LIN {X 0,Y 256.282,Z 675.842,A -85,B 0,C 180,E1 -18466.303,E2 -18466.303} C_VEL
LIN {X 0,Y 258.512,Z 670.213,A -85,B 0,C 180,E1 -18469.867,E2 -18469.867} C_VEL
LIN {X 0,Y 261.173,Z 664.065,A -85,B 0,C 180,E1 -18472.966,E2 -18472.966} C_VEL
LIN {X 0,Y 264.928,Z 655.56,A -85,B 0,C 180,E1 -18476.382,E2 -18476.382} C_VEL
LIN {X 0,Y 269.071,Z 646.458,A -85,B 0,C 180,E1 -18479.324,E2 -18479.324} C_VEL
LIN {X 0,Y 273.55,Z 636.336,A -85,B 0,C 180,E1 -18482.025,E2 -18482.025} C_VEL
LIN {X 0,Y 278.615,Z 624.618,A -85,B 0,C 180,E1 -18484.58,E2 -18484.58} C_VEL
LIN {X 0,Y 283.109,Z 613.564,A -85,B 0,C 180,E1 -18486.569,E2 -18486.569} C_VEL
LIN {X 0,Y 287.912,Z 600.645,A -85,B 0,C 180,E1 -18488.505,E2 -18488.505} C_VEL
LIN {X 0,Y 292.653,Z 586.785,A -85,B 0,C 180,E1 -18490.196,E2 -18490.196} C_VEL
LIN {X 0,Y 296.833,Z 573.328,A -85,B 0,C 180,E1 -18491.525,E2 -18491.525} C_VEL
LIN {X 0,Y 300.553,Z 558.842,A -85,B 0,C 180,E1 -18492.697,E2 -18492.697} C_VEL
LIN {X 0,Y 303.97,Z 543.205,A -85,B 0,C 180,E1 -18493.688,E2 -18493.688} C_VEL
LIN {X 0,Y 306.838,Z 526.737,A -85,B 0,C 180,E1 -18494.466,E2 -18494.466} C_VEL
LIN {X 0,Y 308.914,Z 510.285,A -85,B 0,C 180,E1 -18495.012,E2 -18495.012} C_VEL
LIN {X 0,Y 316.401,Z 389.403,A -85,B 0,C 180,E1 -18497.751,E2 -18497.751} C_VEL
LIN {X 0,Y 310.716,Z 378.003,A -85,B 0,C 180,E1 -18499.592,E2 -18499.592} C_VEL
LIN {X 0,Y 304.506,Z 366.741,A -85,B 0,C 180,E1 -18501.741,E2 -18501.741} C_VEL
LIN {X 0,Y 298.717,Z 357.161,A -85,B 0,C 180,E1 -18503.921,E2 -18503.921} C_VEL
LIN {X 0,Y 292.889,Z 347.944,A -85,B 0,C 180,E1 -18506.349,E2 -18506.349} C_VEL
LIN {X 0,Y 289.275,Z 342.774,A -85,B 0,C 180,E1 -18507.981,E2 -18507.981} C_VEL
LIN {X 0,Y 285.853,Z 337.855,A -85,B 0,C 180,E1 -18509.676,E2 -18509.676} C_VEL
LIN {X 0,Y 281.014,Z 331.224,A -85,B 0,C 180,E1 -18512.335,E2 -18512.335} C_VEL
LIN {X 0,Y 278.285,Z 328.209,A -85,B 0,C 180,E1 -18513.973,E2 -18513.973} C_VEL
LIN {X 0,Y 277.263,Z 326.406,A -85,B 0,C 180,E1 -18514.686,E2 -18514.686} C_VEL
LIN {X 0,Y 274.465,Z 324.032,A -85,B 0,C 180,E1 -18516.597,E2 -18516.597} C_VEL
LIN {X 0,Y 272.679,Z 320.875,A -85,B 0,C 180,E1 -18518.104,E2 -18518.104} C_VEL
LIN {X 0,Y 269.81,Z 318.889,A -85,B 0,C 180,E1 -18520.579,E2 -18520.579} C_VEL
LIN {X 0,Y 268.115,Z 316.082,A -85,B 0,C 180,E1 -18522.567,E2 -18522.567} C_VEL
LIN {X 0,Y 267.662,Z 314.997,A -85,B 0,C 180,E1 -18523.213,E2 -18523.213} C_VEL
LIN {X 0,Y 263.908,Z 312.436,A -85,B 0,C 180,E1 -18530.033,E2 -18530.033} C_VEL
LIN {X 0,Y 263.493,Z 311.642,A -85,B 0,C 180,E1 -18532.337,E2 -18532.337} C_VEL
LIN {X 0,Y 263.433,Z 311.699,A -85,B 0,C 180,E1 -18534.643,E2 -18534.643} C_VEL
LIN {X 0,Y 264.572,Z 312.819,A -85,B 0,C 180,E1 -18539.24,E2 -18539.24} C_VEL
LIN {X 0,Y 268.053,Z 315.309,A -85,B 0,C 180,E1 -18544.706,E2 -18544.706} C_VEL
LIN {X 0,Y 269.415,Z 318.063,A -85,B 0,C 180,E1 -18546.413,E2 -18546.413} C_VEL
LIN {X 0,Y 272.147,Z 320.485,A -85,B 0,C 180,E1 -18548.914,E2 -18548.914} C_VEL
LIN {X 0,Y 272.948,Z 321.205,A -85,B 0,C 180,E1 -18549.565,E2 -18549.565} C_VEL
LIN {X 0,Y 274.825,Z 324.302,A -85,B 0,C 180,E1 -18551.105,E2 -18551.105} C_VEL
LIN {X 0,Y 277.54,Z 326.712,A -85,B 0,C 180,E1 -18552.942,E2 -18552.942} C_VEL
LIN {X 0,Y 279.846,Z 330.125,A -85,B 0,C 180,E1 -18554.441,E2 -18554.441} C_VEL
LIN {X 0,Y 281.946,Z 332.247,A -85,B 0,C 180,E1 -18555.636,E2 -18555.636} C_VEL
LIN {X 0,Y 284.858,Z 335.997,A -85,B 0,C 180,E1 -18557.222,E2 -18557.222} C_VEL
LIN {X 0,Y 286.192,Z 337.735,A -85,B 0,C 180,E1 -18557.908,E2 -18557.908} C_VEL
LIN {X 0,Y 290.002,Z 342.639,A -85,B 0,C 180,E1 -18559.742,E2 -18559.742} C_VEL
LIN {X 0,Y 294.08,Z 348.095,A -85,B 0,C 180,E1 -18561.53,E2 -18561.53} C_VEL
LIN {X 0,Y 299.43,Z 355.459,A -85,B 0,C 180,E1 -18563.674,E2 -18563.674} C_VEL
LIN {X 0,Y 306.714,Z 366.264,A -85,B 0,C 180,E1 -18566.307,E2 -18566.307} C_VEL
LIN {X 0,Y 313.655,Z 377.566,A -85,B 0,C 180,E1 -18568.583,E2 -18568.583} C_VEL
LIN {X 0,Y 316.643,Z 382.91,A -85,B 0,C 180,E1 -18569.512,E2 -18569.512} C_VEL
LIN {X 0,Y 315.495,Z 402.823,A -85,B 0,C 180,E1 -18569.977,E2 -18569.977} C_VEL
LIN {X 0,Y 309.458,Z 498.844,A -85,B 0,C 180,E1 -18572.149,E2 -18572.149} C_VEL
LIN {X 0,Y 307.487,Z 515.059,A -85,B 0,C 180,E1 -18572.712,E2 -18572.712} C_VEL
LIN {X 0,Y 304.889,Z 531.096,A -85,B 0,C 180,E1 -18573.517,E2 -18573.517} C_VEL
LIN {X 0,Y 301.499,Z 547.393,A -85,B 0,C 180,E1 -18574.599,E2 -18574.599} C_VEL
LIN {X 0,Y 297.861,Z 561.75,A -85,B 0,C 180,E1 -18575.799,E2 -18575.799} C_VEL
LIN {X 0,Y 293.557,Z 576.25,A -85,B 0,C 180,E1 -18577.304,E2 -18577.304} C_VEL
LIN {X 0,Y 289.209,Z 589.149,A -85,B 0,C 180,E1 -18578.956,E2 -18578.956} C_VEL
LIN {X 0,Y 284.196,Z 602.561,A -85,B 0,C 180,E1 -18581.04,E2 -18581.04} C_VEL
LIN {X 0,Y 279.535,Z 613.986,A -85,B 0,C 180,E1 -18583.188,E2 -18583.188} C_VEL
LIN {X 0,Y 274.591,Z 625.334,A -85,B 0,C 180,E1 -18585.779,E2 -18585.779} C_VEL
LIN {X 0,Y 270.165,Z 634.852,A -85,B 0,C 180,E1 -18588.444,E2 -18588.444} C_VEL
LIN {X 0,Y 266.327,Z 642.967,A -85,B 0,C 180,E1 -18591.19,E2 -18591.19} C_VEL
LIN {X 0,Y 263.087,Z 649.861,A -85,B 0,C 180,E1 -18594.006,E2 -18594.006} C_VEL
LIN {X 0,Y 260.017,Z 656.29,A -85,B 0,C 180,E1 -18597.277,E2 -18597.277} C_VEL
LIN {X 0,Y 257.501,Z 661.786,A -85,B 0,C 180,E1 -18600.856,E2 -18600.856} C_VEL
LIN {X 0,Y 255.936,Z 665.412,A -85,B 0,C 180,E1 -18603.937,E2 -18603.937} C_VEL
LIN {X 0,Y 254.774,Z 668.176,A -85,B 0,C 180,E1 -18607.282,E2 -18607.282} C_VEL
LIN {X 0,Y 254.125,Z 669.944,A -85,B 0,C 180,E1 -18610.618,E2 -18610.618} C_VEL
LIN {X 0,Y 253.789,Z 670.613,A -85,B 0,C 180,E1 -18613.923,E2 -18613.923} C_VEL
LIN {X 0,Y 253.738,Z 670.334,A -85,B 0,C 180,E1 -18617.198,E2 -18617.198} C_VEL
LIN {X 0,Y 253.774,Z 669.044,A -85,B 0,C 180,E1 -18620.435,E2 -18620.435} C_VEL
LIN {X 0,Y 254.305,Z 666.26,A -85,B 0,C 180,E1 -18624.221,E2 -18624.221} C_VEL
LIN {X 0,Y 254.766,Z 662.566,A -85,B 0,C 180,E1 -18627.628,E2 -18627.628} C_VEL
LIN {X 0,Y 255.672,Z 657.991,A -85,B 0,C 180,E1 -18630.787,E2 -18630.787} C_VEL
LIN {X 0,Y 257.085,Z 652.288,A -85,B 0,C 180,E1 -18633.919,E2 -18633.919} C_VEL
LIN {X 0,Y 258.941,Z 645.419,A -85,B 0,C 180,E1 -18637.015,E2 -18637.015} C_VEL
LIN {X 0,Y 261.842,Z 635.962,A -85,B 0,C 180,E1 -18640.438,E2 -18640.438} C_VEL
LIN {X 0,Y 265.051,Z 625.811,A -85,B 0,C 180,E1 -18643.415,E2 -18643.415} C_VEL
LIN {X 0,Y 268.266,Z 615.356,A -85,B 0,C 180,E1 -18645.966,E2 -18645.966} C_VEL
LIN {X 0,Y 271.802,Z 603.133,A -85,B 0,C 180,E1 -18648.466,E2 -18648.466} C_VEL
LIN {X 0,Y 275.208,Z 590.86,A -85,B 0,C 180,E1 -18650.557,E2 -18650.557} C_VEL
LIN {X 0,Y 278.588,Z 577.562,A -85,B 0,C 180,E1 -18652.43,E2 -18652.43} C_VEL
LIN {X 0,Y 281.942,Z 563.146,A -85,B 0,C 180,E1 -18654.09,E2 -18654.09} C_VEL
LIN {X 0,Y 284.627,Z 549.4,A -85,B 0,C 180,E1 -18655.405,E2 -18655.405} C_VEL
LIN {X 0,Y 286.727,Z 536.983,A -85,B 0,C 180,E1 -18656.376,E2 -18656.376} C_VEL
LIN {X 0,Y 289.155,Z 520.691,A -85,B 0,C 180,E1 -18657.356,E2 -18657.356} C_VEL
LIN {X 0,Y 290.872,Z 504.966,A -85,B 0,C 180,E1 -18658.06,E2 -18658.06} C_VEL
LIN {X 0,Y 292.168,Z 487.884,A -85,B 0,C 180,E1 -18658.56,E2 -18658.56} C_VEL
LIN {X 0,Y 297.829,Z 371.285,A -85,B 0,C 180,E1 -18661.275,E2 -18661.275} C_VEL
LIN {X 0,Y 297.355,Z 369.401,A -85,B 0,C 180,E1 -18661.409,E2 -18661.409} C_VEL
LIN {X 0,Y 291.594,Z 358.102,A -85,B 0,C 180,E1 -18662.726,E2 -18662.726} C_VEL
LIN {X 0,Y 282.106,Z 341.691,A -85,B 0,C 180,E1 -18664.988,E2 -18664.988} C_VEL
LIN {X 0,Y 273.66,Z 328.4,A -85,B 0,C 180,E1 -18667.161,E2 -18667.161} C_VEL
LIN {X 0,Y 265.648,Z 316.865,A -85,B 0,C 180,E1 -18669.382,E2 -18669.382} C_VEL
LIN {X 0,Y 262.439,Z 312.49,A -85,B 0,C 180,E1 -18670.328,E2 -18670.328} C_VEL
LIN {X 0,Y 260.022,Z 309.315,A -85,B 0,C 180,E1 -18671.062,E2 -18671.062} C_VEL
LIN {X 0,Y 259.132,Z 307.907,A -85,B 0,C 180,E1 -18671.349,E2 -18671.349} C_VEL
LIN {X 0,Y 256.924,Z 305.562,A -85,B 0,C 180,E1 -18672.024,E2 -18672.024} C_VEL
LIN {X 0,Y 256.02,Z 302.892,A -85,B 0,C 180,E1 -18672.413,E2 -18672.413} C_VEL
LIN {X 0,Y 256.005,Z 302.89,A -85,B 0,C 180,E1 -18676.66,E2 -18676.66} C_VEL
LIN {X 0,Y 256.044,Z 302.866,A -85,B 0,C 180,E1 -18680.852,E2 -18680.852} C_VEL
LIN {X 0,Y 256.042,Z 302.843,A -85,B 0,C 180,E1 -18682.1,E2 -18682.1} C_VEL
LIN {X 0,Y 255.418,Z 302.915,A -85,B 0,C 180,E1 -18683.412,E2 -18683.412} C_VEL
LIN {X 0,Y 252.558,Z 303.294,A -85,B 0,C 180,E1 -18685.55,E2 -18685.55} C_VEL
LIN {X 0,Y 250.108,Z 303.636,A -85,B 0,C 180,E1 -18687.29,E2 -18687.29} C_VEL
LIN {X 0,Y 249.065,Z 303.772,A -85,B 0,C 180,E1 -18688.641,E2 -18688.641} C_VEL
LIN {X 0,Y 248.987,Z 303.771,A -85,B 0,C 180,E1 -18689.099,E2 -18689.099} C_VEL
LIN {X 0,Y 249.031,Z 303.776,A -85,B 0,C 180,E1 -18693.156,E2 -18693.156} C_VEL
LIN {X 0,Y 249.055,Z 303.753,A -85,B 0,C 180,E1 -18696.729,E2 -18696.729} C_VEL
LIN {X 0,Y 249.087,Z 303.765,A -85,B 0,C 180,E1 -18700.209,E2 -18700.209} C_VEL
LIN {X 0,Y 249.197,Z 303.744,A -85,B 0,C 180,E1 -18703.618,E2 -18703.618} C_VEL
LIN {X 0,Y 249.244,Z 303.728,A -85,B 0,C 180,E1 -18708.615,E2 -18708.615} C_VEL
LIN {X 0,Y 249.445,Z 303.723,A -85,B 0,C 180,E1 -18711.901,E2 -18711.901} C_VEL
LIN {X 0,Y 249.279,Z 303.725,A -85,B 0,C 180,E1 -18715.147,E2 -18715.147} C_VEL
LIN {X 0,Y 249.672,Z 303.691,A -85,B 0,C 180,E1 -18718.386,E2 -18718.386} C_VEL
LIN {X 0,Y 249.675,Z 303.679,A -85,B 0,C 180,E1 -18721.612,E2 -18721.612} C_VEL
LIN {X 0,Y 249.449,Z 303.691,A -85,B 0,C 180,E1 -18726.47,E2 -18726.47} C_VEL
LIN {X 0,Y 249.343,Z 303.732,A -85,B 0,C 180,E1 -18729.736,E2 -18729.736} C_VEL
LIN {X 0,Y 249.183,Z 303.759,A -85,B 0,C 180,E1 -18734.704,E2 -18734.704} C_VEL
LIN {X 0,Y 249.12,Z 303.767,A -85,B 0,C 180,E1 -18738.078,E2 -18738.078} C_VEL
LIN {X 0,Y 249.086,Z 303.769,A -85,B 0,C 180,E1 -18741.517,E2 -18741.517} C_VEL
LIN {X 0,Y 249.129,Z 303.763,A -85,B 0,C 180,E1 -18745.481,E2 -18745.481} C_VEL
LIN {X 0,Y 249.079,Z 303.772,A -85,B 0,C 180,E1 -18748.991,E2 -18748.991} C_VEL
LIN {X 0,Y 249.026,Z 303.779,A -85,B 0,C 180,E1 -18752.285,E2 -18752.285} C_VEL
LIN {X 0,Y 249.973,Z 306.545,A -85,B 0,C 180,E1 -18752.706,E2 -18752.706} C_VEL
LIN {X 0,Y 252.086,Z 308.765,A -85,B 0,C 180,E1 -18753.408,E2 -18753.408} C_VEL
LIN {X 0,Y 252.84,Z 309.519,A -85,B 0,C 180,E1 -18753.654,E2 -18753.654} C_VEL
LIN {X 0,Y 254.89,Z 312.734,A -85,B 0,C 180,E1 -18754.358,E2 -18754.358} C_VEL
LIN {X 0,Y 256.51,Z 314.52,A -85,B 0,C 180,E1 -18754.867,E2 -18754.867} C_VEL
LIN {X 0,Y 259.22,Z 318.185,A -85,B 0,C 180,E1 -18755.722,E2 -18755.722} C_VEL
LIN {X 0,Y 264.025,Z 325.444,A -85,B 0,C 180,E1 -18757.19,E2 -18757.19} C_VEL
LIN {X 0,Y 270.599,Z 336.395,A -85,B 0,C 180,E1 -18759.096,E2 -18759.096} C_VEL
LIN {X 0,Y 278.225,Z 350.18,A -85,B 0,C 180,E1 -18761.173,E2 -18761.173} C_VEL
LIN {X 0,Y 285.454,Z 364.869,A -85,B 0,C 180,E1 -18763.034,E2 -18763.034} C_VEL
LIN {X 0,Y 292.165,Z 379.915,A -85,B 0,C 180,E1 -18764.686,E2 -18764.686} C_VEL
LIN {X 0,Y 285.516,Z 510.664,A -85,B 0,C 180,E1 -18767.806,E2 -18767.806} C_VEL
LIN {X 0,Y 283.759,Z 527.699,A -85,B 0,C 180,E1 -18768.448,E2 -18768.448} C_VEL
LIN {X 0,Y 281.493,Z 543.45,A -85,B 0,C 180,E1 -18769.288,E2 -18769.288} C_VEL
LIN {X 0,Y 278.588,Z 559.632,A -85,B 0,C 180,E1 -18770.433,E2 -18770.433} C_VEL
LIN {X 0,Y 275.831,Z 572.821,A -85,B 0,C 180,E1 -18771.607,E2 -18771.607} C_VEL
LIN {X 0,Y 272.213,Z 587.811,A -85,B 0,C 180,E1 -18773.263,E2 -18773.263} C_VEL
LIN {X 0,Y 268.642,Z 601.267,A -85,B 0,C 180,E1 -18775.091,E2 -18775.091} C_VEL
LIN {X 0,Y 265.222,Z 613.539,A -85,B 0,C 180,E1 -18777.097,E2 -18777.097} C_VEL
LIN {X 0,Y 261.658,Z 624.974,A -85,B 0,C 180,E1 -18779.314,E2 -18779.314} C_VEL
LIN {X 0,Y 258.167,Z 636.389,A -85,B 0,C 180,E1 -18781.992,E2 -18781.992} C_VEL
LIN {X 0,Y 255.048,Z 646.135,A -85,B 0,C 180,E1 -18784.716,E2 -18784.716} C_VEL
LIN {X 0,Y 252.296,Z 655.591,A -85,B 0,C 180,E1 -18787.91,E2 -18787.91} C_VEL
LIN {X 0,Y 250.074,Z 663.425,A -85,B 0,C 180,E1 -18791.144,E2 -18791.144} C_VEL
LIN {X 0,Y 248.522,Z 670.114,A -85,B 0,C 180,E1 -18794.558,E2 -18794.558} C_VEL
LIN {X 0,Y 247.555,Z 675.124,A -85,B 0,C 180,E1 -18797.707,E2 -18797.707} C_VEL
LIN {X 0,Y 247.097,Z 678.259,A -85,B 0,C 180,E1 -18800.174,E2 -18800.174} C_VEL
LIN {X 0,Y 246.938,Z 681.534,A -85,B 0,C 180,E1 -18803.463,E2 -18803.463} C_VEL
LIN {X 0,Y 246.885,Z 683.72,A -85,B 0,C 180,E1 -18806.736,E2 -18806.736} C_VEL
LIN {X 0,Y 246.981,Z 684.942,A -85,B 0,C 180,E1 -18810,E2 -18810} C_VEL
LIN {X 0,Y 246.837,Z 685.129,A -85,B 0,C 180,E1 -18813.265,E2 -18813.265} C_VEL
LIN {X 0,Y 246.86,Z 684.395,A -85,B 0,C 180,E1 -18816.539,E2 -18816.539} C_VEL
LIN {X 0,Y 247.156,Z 682.668,A -85,B 0,C 180,E1 -18819.824,E2 -18819.824} C_VEL
LIN {X 0,Y 247.92,Z 680.007,A -85,B 0,C 180,E1 -18823.108,E2 -18823.108} C_VEL
LIN {X 0,Y 249.271,Z 676.096,A -85,B 0,C 180,E1 -18826.547,E2 -18826.547} C_VEL
LIN {X 0,Y 251.161,Z 671.616,A -85,B 0,C 180,E1 -18829.621,E2 -18829.621} C_VEL
LIN {X 0,Y 253.819,Z 665.734,A -85,B 0,C 180,E1 -18832.808,E2 -18832.808} C_VEL
LIN {X 0,Y 257.555,Z 657.691,A -85,B 0,C 180,E1 -18836.322,E2 -18836.322} C_VEL
LIN {X 0,Y 261.714,Z 649.102,A -85,B 0,C 180,E1 -18839.346,E2 -18839.346} C_VEL
LIN {X 0,Y 266.735,Z 638.415,A -85,B 0,C 180,E1 -18842.392,E2 -18842.392} C_VEL
LIN {X 0,Y 272.066,Z 626.675,A -85,B 0,C 180,E1 -18845.083,E2 -18845.083} C_VEL
LIN {X 0,Y 276.631,Z 615.951,A -85,B 0,C 180,E1 -18847.113,E2 -18847.113} C_VEL
LIN {X 0,Y 281.946,Z 602.57,A -85,B 0,C 180,E1 -18849.209,E2 -18849.209} C_VEL
LIN {X 0,Y 286.428,Z 590.233,A -85,B 0,C 180,E1 -18850.79,E2 -18850.79} C_VEL
LIN {X 0,Y 291.079,Z 575.761,A -85,B 0,C 180,E1 -18852.302,E2 -18852.302} C_VEL
LIN {X 0,Y 295.442,Z 559.974,A -85,B 0,C 180,E1 -18853.619,E2 -18853.619} C_VEL
LIN {X 0,Y 298.693,Z 546.026,A -85,B 0,C 180,E1 -18854.545,E2 -18854.545} C_VEL
LIN {X 0,Y 301.828,Z 529.373,A -85,B 0,C 180,E1 -18855.376,E2 -18855.376} C_VEL
LIN {X 0,Y 304.023,Z 513.672,A -85,B 0,C 180,E1 -18855.918,E2 -18855.918} C_VEL
LIN {X 0,Y 305.657,Z 491.795,A -85,B 0,C 180,E1 -18856.48,E2 -18856.48} C_VEL
LIN {X 0,Y 311.962,Z 392.471,A -85,B 0,C 180,E1 -18858.712,E2 -18858.712} C_VEL
LIN {X 0,Y 306.688,Z 381.757,A -85,B 0,C 180,E1 -18860.508,E2 -18860.508} C_VEL
LIN {X 0,Y 300.287,Z 370.018,A -85,B 0,C 180,E1 -18862.844,E2 -18862.844} C_VEL
LIN {X 0,Y 294.471,Z 360.375,A -85,B 0,C 180,E1 -18865.173,E2 -18865.173} C_VEL
LIN {X 0,Y 289.954,Z 353.204,A -85,B 0,C 180,E1 -18867.158,E2 -18867.158} C_VEL
LIN {X 0,Y 287.239,Z 349.171,A -85,B 0,C 180,E1 -18868.442,E2 -18868.442} C_VEL
LIN {X 0,Y 283.9,Z 344.285,A -85,B 0,C 180,E1 -18870.147,E2 -18870.147} C_VEL
LIN {X 0,Y 279.285,Z 337.821,A -85,B 0,C 180,E1 -18872.764,E2 -18872.764} C_VEL
LIN {X 0,Y 276.497,Z 334.578,A -85,B 0,C 180,E1 -18874.505,E2 -18874.505} C_VEL
LIN {X 0,Y 275.556,Z 333.045,A -85,B 0,C 180,E1 -18875.176,E2 -18875.176} C_VEL
LIN {X 0,Y 272.747,Z 330.381,A -85,B 0,C 180,E1 -18877.191,E2 -18877.191} C_VEL
LIN {X 0,Y 271.223,Z 327.703,A -85,B 0,C 180,E1 -18878.525,E2 -18878.525} C_VEL
LIN {X 0,Y 268.356,Z 325.445,A -85,B 0,C 180,E1 -18881.14,E2 -18881.14} C_VEL
LIN {X 0,Y 266.807,Z 322.608,A -85,B 0,C 180,E1 -18883.09,E2 -18883.09} C_VEL
LIN {X 0,Y 266.581,Z 321.964,A -85,B 0,C 180,E1 -18883.44,E2 -18883.44} C_VEL
LIN {X 0,Y 262.982,Z 319.422,A -85,B 0,C 180,E1 -18890.208,E2 -18890.208} C_VEL
LIN {X 0,Y 262.617,Z 318.699,A -85,B 0,C 180,E1 -18892.311,E2 -18892.311} C_VEL
LIN {X 0,Y 262.557,Z 318.73,A -85,B 0,C 180,E1 -18894.625,E2 -18894.625} C_VEL
LIN {X 0,Y 263.687,Z 319.881,A -85,B 0,C 180,E1 -18899.237,E2 -18899.237} C_VEL
LIN {X 0,Y 266.881,Z 322.267,A -85,B 0,C 180,E1 -18904.389,E2 -18904.389} C_VEL
LIN {X 0,Y 268.387,Z 325.133,A -85,B 0,C 180,E1 -18906.296,E2 -18906.296} C_VEL
LIN {X 0,Y 271.018,Z 327.446,A -85,B 0,C 180,E1 -18908.741,E2 -18908.741} C_VEL
LIN {X 0,Y 271.498,Z 327.944,A -85,B 0,C 180,E1 -18909.147,E2 -18909.147} C_VEL
LIN {X 0,Y 273.536,Z 331.203,A -85,B 0,C 180,E1 -18910.853,E2 -18910.853} C_VEL
LIN {X 0,Y 275.971,Z 333.473,A -85,B 0,C 180,E1 -18912.549,E2 -18912.549} C_VEL
LIN {X 0,Y 278.466,Z 337.018,A -85,B 0,C 180,E1 -18914.199,E2 -18914.199} C_VEL
LIN {X 0,Y 280.138,Z 338.785,A -85,B 0,C 180,E1 -18915.179,E2 -18915.179} C_VEL
LIN {X 0,Y 283.249,Z 342.749,A -85,B 0,C 180,E1 -18916.912,E2 -18916.912} C_VEL
LIN {X 0,Y 287.981,Z 349.137,A -85,B 0,C 180,E1 -18919.3,E2 -18919.3} C_VEL
LIN {X 0,Y 292.559,Z 355.305,A -85,B 0,C 180,E1 -18921.353,E2 -18921.353} C_VEL
LIN {X 0,Y 299.18,Z 364.828,A -85,B 0,C 180,E1 -18924.025,E2 -18924.025} C_VEL
LIN {X 0,Y 306.111,Z 375.653,A -85,B 0,C 180,E1 -18926.53,E2 -18926.53} C_VEL
LIN {X 0,Y 312.261,Z 386.159,A -85,B 0,C 180,E1 -18928.565,E2 -18928.565} C_VEL
LIN {X 0,Y 304.942,Z 498.932,A -85,B 0,C 180,E1 -18931.126,E2 -18931.126} C_VEL
LIN {X 0,Y 302.876,Z 515.219,A -85,B 0,C 180,E1 -18931.685,E2 -18931.685} C_VEL
LIN {X 0,Y 300.358,Z 530.516,A -85,B 0,C 180,E1 -18932.454,E2 -18932.454} C_VEL
LIN {X 0,Y 297.394,Z 544.888,A -85,B 0,C 180,E1 -18933.385,E2 -18933.385} C_VEL
LIN {X 0,Y 294.011,Z 558.094,A -85,B 0,C 180,E1 -18934.443,E2 -18934.443} C_VEL
LIN {X 0,Y 289.61,Z 572.976,A -85,B 0,C 180,E1 -18935.919,E2 -18935.919} C_VEL
LIN {X 0,Y 284.973,Z 586.716,A -85,B 0,C 180,E1 -18937.602,E2 -18937.602} C_VEL
LIN {X 0,Y 280.132,Z 599.542,A -85,B 0,C 180,E1 -18939.514,E2 -18939.514} C_VEL
LIN {X 0,Y 274.408,Z 613.211,A -85,B 0,C 180,E1 -18942.035,E2 -18942.035} C_VEL
LIN {X 0,Y 269.135,Z 624.8,A -85,B 0,C 180,E1 -18944.689,E2 -18944.689} C_VEL
LIN {X 0,Y 264.526,Z 634.308,A -85,B 0,C 180,E1 -18947.352,E2 -18947.352} C_VEL
LIN {X 0,Y 259.896,Z 643.608,A -85,B 0,C 180,E1 -18950.544,E2 -18950.544} C_VEL
LIN {X 0,Y 256.07,Z 651.292,A -85,B 0,C 180,E1 -18953.837,E2 -18953.837} C_VEL
LIN {X 0,Y 252.928,Z 657.539,A -85,B 0,C 180,E1 -18957.191,E2 -18957.191} C_VEL
LIN {X 0,Y 250.04,Z 663.516,A -85,B 0,C 180,E1 -18961.456,E2 -18961.456} C_VEL
LIN {X 0,Y 248.499,Z 666.914,A -85,B 0,C 180,E1 -18964.898,E2 -18964.898} C_VEL
LIN {X 0,Y 247.442,Z 669.272,A -85,B 0,C 180,E1 -18968.331,E2 -18968.331} C_VEL
LIN {X 0,Y 246.86,Z 670.552,A -85,B 0,C 180,E1 -18971.75,E2 -18971.75} C_VEL
LIN {X 0,Y 246.689,Z 670.77,A -85,B 0,C 180,E1 -18975.616,E2 -18975.616} C_VEL
LIN {X 0,Y 246.63,Z 670.118,A -85,B 0,C 180,E1 -18978.494,E2 -18978.494} C_VEL
LIN {X 0,Y 246.799,Z 668.406,A -85,B 0,C 180,E1 -18981.814,E2 -18981.814} C_VEL
LIN {X 0,Y 247.291,Z 665.747,A -85,B 0,C 180,E1 -18985.109,E2 -18985.109} C_VEL
LIN {X 0,Y 248.112,Z 660.959,A -85,B 0,C 180,E1 -18989.188,E2 -18989.188} C_VEL
LIN {X 0,Y 249.236,Z 655.904,A -85,B 0,C 180,E1 -18992.424,E2 -18992.424} C_VEL
LIN {X 0,Y 250.922,Z 649.748,A -85,B 0,C 180,E1 -18995.626,E2 -18995.626} C_VEL
LIN {X 0,Y 253.494,Z 641.227,A -85,B 0,C 180,E1 -18999.173,E2 -18999.173} C_VEL
LIN {X 0,Y 256.533,Z 632.019,A -85,B 0,C 180,E1 -19002.258,E2 -19002.258} C_VEL
LIN {X 0,Y 259.573,Z 622.575,A -85,B 0,C 180,E1 -19004.905,E2 -19004.905} C_VEL
LIN {X 0,Y 263.032,Z 611.599,A -85,B 0,C 180,E1 -19007.493,E2 -19007.493} C_VEL
LIN {X 0,Y 266.843,Z 598.664,A -85,B 0,C 180,E1 -19010.022,E2 -19010.022} C_VEL
LIN {X 0,Y 270.777,Z 584.323,A -85,B 0,C 180,E1 -19012.308,E2 -19012.308} C_VEL
LIN {X 0,Y 274.498,Z 569.698,A -85,B 0,C 180,E1 -19014.183,E2 -19014.183} C_VEL
LIN {X 0,Y 277.646,Z 555.32,A -85,B 0,C 180,E1 -19015.689,E2 -19015.689} C_VEL
LIN {X 0,Y 280.462,Z 539.768,A -85,B 0,C 180,E1 -19017.013,E2 -19017.013} C_VEL
LIN {X 0,Y 283.069,Z 523.613,A -85,B 0,C 180,E1 -19018.046,E2 -19018.046} C_VEL
LIN {X 0,Y 284.941,Z 507.968,A -85,B 0,C 180,E1 -19018.799,E2 -19018.799} C_VEL
LIN {X 0,Y 286.357,Z 490.663,A -85,B 0,C 180,E1 -19019.346,E2 -19019.346} C_VEL
LIN {X 0,Y 292.312,Z 373.29,A -85,B 0,C 180,E1 -19022.116,E2 -19022.116} C_VEL
LIN {X 0,Y 291.273,Z 370.526,A -85,B 0,C 180,E1 -19022.38,E2 -19022.38} C_VEL
LIN {X 0,Y 282.881,Z 354.95,A -85,B 0,C 180,E1 -19024.386,E2 -19024.386} C_VEL
LIN {X 0,Y 274.315,Z 340.56,A -85,B 0,C 180,E1 -19026.578,E2 -19026.578} C_VEL
LIN {X 0,Y 266.456,Z 328.649,A -85,B 0,C 180,E1 -19028.733,E2 -19028.733} C_VEL
LIN {X 0,Y 261.558,Z 321.663,A -85,B 0,C 180,E1 -19030.17,E2 -19030.17} C_VEL
LIN {X 0,Y 258.607,Z 317.645,A -85,B 0,C 180,E1 -19031.074,E2 -19031.074} C_VEL
LIN {X 0,Y 255.546,Z 313.467,A -85,B 0,C 180,E1 -19032.049,E2 -19032.049} C_VEL
LIN {X 0,Y 253.243,Z 310.556,A -85,B 0,C 180,E1 -19032.8,E2 -19032.8} C_VEL
LIN {X 0,Y 252.259,Z 308.92,A -85,B 0,C 180,E1 -19033.146,E2 -19033.146} C_VEL
LIN {X 0,Y 250.137,Z 306.89,A -85,B 0,C 180,E1 -19033.842,E2 -19033.842} C_VEL
LIN {X 0,Y 249.05,Z 304.29,A -85,B 0,C 180,E1 -19034.28,E2 -19034.28} C_VEL
LIN {X 0,Y 248.987,Z 303.783,A -85,B 0,C 180,E1 -19034.334,E2 -19034.334} C_VEL
LIN {X 0,Y 248.968,Z 303.77,A -85,B 0,C 180,E1 -19037.351,E2 -19037.351} C_VEL
LIN {X 0,Y 249.004,Z 303.725,A -85,B 0,C 180,E1 -19041.614,E2 -19041.614} C_VEL
LIN {X 0,Y 249.044,Z 303.729,A -85,B 0,C 180,E1 -19045.638,E2 -19045.638} C_VEL
LIN {X 0,Y 248.987,Z 303.771,A -85,B 0,C 180,E1 -19049.099,E2 -19049.099} C_VEL
LIN {X 0,Y 248.354,Z 303.851,A -85,B 0,C 180,E1 -19050.449,E2 -19050.449} C_VEL
LIN {X 0,Y 245.571,Z 304.203,A -85,B 0,C 180,E1 -19052.652,E2 -19052.652} C_VEL
LIN {X 0,Y 242.353,Z 304.593,A -85,B 0,C 180,E1 -19055.367,E2 -19055.367} C_VEL
LIN {X 0,Y 242.006,Z 304.63,A -85,B 0,C 180,E1 -19056.306,E2 -19056.306} C_VEL
LIN {X 0,Y 242.022,Z 304.65,A -85,B 0,C 180,E1 -19059.606,E2 -19059.606} C_VEL
LIN {X 0,Y 242.117,Z 304.621,A -85,B 0,C 180,E1 -19063.315,E2 -19063.315} C_VEL
LIN {X 0,Y 242.155,Z 304.621,A -85,B 0,C 180,E1 -19066.574,E2 -19066.574} C_VEL
LIN {X 0,Y 242.393,Z 304.603,A -85,B 0,C 180,E1 -19071.663,E2 -19071.663} C_VEL
LIN {X 0,Y 242.414,Z 304.58,A -85,B 0,C 180,E1 -19073.34,E2 -19073.34} C_VEL
LIN {X 0,Y 242.632,Z 304.568,A -85,B 0,C 180,E1 -19078.339,E2 -19078.339} C_VEL
LIN {X 0,Y 242.636,Z 304.556,A -85,B 0,C 180,E1 -19081.659,E2 -19081.659} C_VEL
LIN {X 0,Y 242.42,Z 304.565,A -85,B 0,C 180,E1 -19086.658,E2 -19086.658} C_VEL
LIN {X 0,Y 242.267,Z 304.617,A -85,B 0,C 180,E1 -19090.023,E2 -19090.023} C_VEL
LIN {X 0,Y 242.139,Z 304.632,A -85,B 0,C 180,E1 -19095.142,E2 -19095.142} C_VEL
LIN {X 0,Y 242.06,Z 304.643,A -85,B 0,C 180,E1 -19098.624,E2 -19098.624} C_VEL
LIN {X 0,Y 242.012,Z 304.648,A -85,B 0,C 180,E1 -19102.179,E2 -19102.179} C_VEL
LIN {X 0,Y 242.065,Z 304.644,A -85,B 0,C 180,E1 -19105.837,E2 -19105.837} C_VEL
LIN {X 0,Y 242.036,Z 304.762,A -85,B 0,C 180,E1 -19110.178,E2 -19110.178} C_VEL
LIN {X 0,Y 242.925,Z 307.374,A -85,B 0,C 180,E1 -19110.596,E2 -19110.596} C_VEL
LIN {X 0,Y 244.938,Z 309.582,A -85,B 0,C 180,E1 -19111.34,E2 -19111.34} C_VEL
LIN {X 0,Y 245.808,Z 310.35,A -85,B 0,C 180,E1 -19111.645,E2 -19111.645} C_VEL
LIN {X 0,Y 247.802,Z 313.526,A -85,B 0,C 180,E1 -19112.393,E2 -19112.393} C_VEL
LIN {X 0,Y 249.717,Z 315.553,A -85,B 0,C 180,E1 -19113.043,E2 -19113.043} C_VEL
LIN {X 0,Y 252.394,Z 319.214,A -85,B 0,C 180,E1 -19113.961,E2 -19113.961} C_VEL
LIN {X 0,Y 257.381,Z 326.144,A -85,B 0,C 180,E1 -19115.587,E2 -19115.587} C_VEL
LIN {X 0,Y 260.923,Z 331.688,A -85,B 0,C 180,E1 -19116.699,E2 -19116.699} C_VEL
LIN {X 0,Y 266.071,Z 340.378,A -85,B 0,C 180,E1 -19118.248,E2 -19118.248} C_VEL
LIN {X 0,Y 273.311,Z 353.584,A -85,B 0,C 180,E1 -19120.305,E2 -19120.305} C_VEL
LIN {X 0,Y 280.528,Z 368.263,A -85,B 0,C 180,E1 -19122.245,E2 -19122.245} C_VEL
LIN {X 0,Y 286.652,Z 382.108,A -85,B 0,C 180,E1 -19123.818,E2 -19123.818} C_VEL
LIN {X 0,Y 279.906,Z 510.628,A -85,B 0,C 180,E1 -19126.927,E2 -19126.927} C_VEL
LIN {X 0,Y 278.085,Z 527.811,A -85,B 0,C 180,E1 -19127.587,E2 -19127.587} C_VEL
LIN {X 0,Y 275.622,Z 544.126,A -85,B 0,C 180,E1 -19128.474,E2 -19128.474} C_VEL
LIN {X 0,Y 272.648,Z 560.104,A -85,B 0,C 180,E1 -19129.636,E2 -19129.636} C_VEL
LIN {X 0,Y 269.808,Z 573.208,A -85,B 0,C 180,E1 -19130.827,E2 -19130.827} C_VEL
LIN {X 0,Y 265.949,Z 588.586,A -85,B 0,C 180,E1 -19132.569,E2 -19132.569} C_VEL
LIN {X 0,Y 262.399,Z 601.463,A -85,B 0,C 180,E1 -19134.371,E2 -19134.371} C_VEL
LIN {X 0,Y 258.516,Z 614.66,A -85,B 0,C 180,E1 -19136.598,E2 -19136.598} C_VEL
LIN {X 0,Y 254.604,Z 626.868,A -85,B 0,C 180,E1 -19139.075,E2 -19139.075} C_VEL
LIN {X 0,Y 251.273,Z 637.192,A -85,B 0,C 180,E1 -19141.609,E2 -19141.609} C_VEL
LIN {X 0,Y 248.105,Z 646.769,A -85,B 0,C 180,E1 -19144.407,E2 -19144.407} C_VEL
LIN {X 0,Y 245.279,Z 656.075,A -85,B 0,C 180,E1 -19147.688,E2 -19147.688} C_VEL
LIN {X 0,Y 243.254,Z 662.917,A -85,B 0,C 180,E1 -19150.595,E2 -19150.595} C_VEL
LIN {X 0,Y 241.602,Z 669.365,A -85,B 0,C 180,E1 -19153.923,E2 -19153.923} C_VEL
LIN {X 0,Y 240.553,Z 674.744,A -85,B 0,C 180,E1 -19157.343,E2 -19157.343} C_VEL
LIN {X 0,Y 239.885,Z 679.724,A -85,B 0,C 180,E1 -19161.577,E2 -19161.577} C_VEL
LIN {X 0,Y 239.837,Z 682.522,A -85,B 0,C 180,E1 -19165.068,E2 -19165.068} C_VEL
LIN {X 0,Y 239.84,Z 684.226,A -85,B 0,C 180,E1 -19168.321,E2 -19168.321} C_VEL
LIN {X 0,Y 239.911,Z 684.698,A -85,B 0,C 180,E1 -19170,E2 -19170} C_VEL
LIN {X 0,Y 239.742,Z 684.933,A -85,B 0,C 180,E1 -19173.361,E2 -19173.361} C_VEL
LIN {X 0,Y 239.772,Z 684.224,A -85,B 0,C 180,E1 -19176.733,E2 -19176.733} C_VEL
LIN {X 0,Y 240.088,Z 682.55,A -85,B 0,C 180,E1 -19180.116,E2 -19180.116} C_VEL
LIN {X 0,Y 240.935,Z 679.917,A -85,B 0,C 180,E1 -19183.495,E2 -19183.495} C_VEL
LIN {X 0,Y 242.757,Z 675.204,A -85,B 0,C 180,E1 -19187.697,E2 -19187.697} C_VEL
LIN {X 0,Y 245.028,Z 670.263,A -85,B 0,C 180,E1 -19191.01,E2 -19191.01} C_VEL
LIN {X 0,Y 247.978,Z 664.177,A -85,B 0,C 180,E1 -19194.265,E2 -19194.265} C_VEL
LIN {X 0,Y 252.158,Z 655.81,A -85,B 0,C 180,E1 -19197.83,E2 -19197.83} C_VEL
LIN {X 0,Y 256.669,Z 646.866,A -85,B 0,C 180,E1 -19200.891,E2 -19200.891} C_VEL
LIN {X 0,Y 261.515,Z 637.024,A -85,B 0,C 180,E1 -19203.658,E2 -19203.658} C_VEL
LIN {X 0,Y 267.006,Z 625.405,A -85,B 0,C 180,E1 -19206.316,E2 -19206.316} C_VEL
LIN {X 0,Y 271.847,Z 614.476,A -85,B 0,C 180,E1 -19208.351,E2 -19208.351} C_VEL
LIN {X 0,Y 277.281,Z 601.017,A -85,B 0,C 180,E1 -19210.44,E2 -19210.44} C_VEL
LIN {X 0,Y 282.488,Z 586.908,A -85,B 0,C 180,E1 -19212.201,E2 -19212.201} C_VEL
LIN {X 0,Y 287.41,Z 571.899,A -85,B 0,C 180,E1 -19213.693,E2 -19213.693} C_VEL
LIN {X 0,Y 291.886,Z 555.272,A -85,B 0,C 180,E1 -19215.015,E2 -19215.015} C_VEL
LIN {X 0,Y 295.6,Z 538.694,A -85,B 0,C 180,E1 -19215.989,E2 -19215.989} C_VEL
LIN {X 0,Y 298.291,Z 522.957,A -85,B 0,C 180,E1 -19216.673,E2 -19216.673} C_VEL
LIN {X 0,Y 300.354,Z 505.518,A -85,B 0,C 180,E1 -19217.199,E2 -19217.199} C_VEL
LIN {X 0,Y 307.576,Z 395.442,A -85,B 0,C 180,E1 -19219.717,E2 -19219.717} C_VEL
LIN {X 0,Y 303.051,Z 386.207,A -85,B 0,C 180,E1 -19221.329,E2 -19221.329} C_VEL
LIN {X 0,Y 297.425,Z 375.64,A -85,B 0,C 180,E1 -19223.478,E2 -19223.478} C_VEL
LIN {X 0,Y 291.759,Z 366.017,A -85,B 0,C 180,E1 -19225.837,E2 -19225.837} C_VEL
LIN {X 0,Y 287.503,Z 359.084,A -85,B 0,C 180,E1 -19227.785,E2 -19227.785} C_VEL
LIN {X 0,Y 284.896,Z 355.157,A -85,B 0,C 180,E1 -19229.07,E2 -19229.07} C_VEL
LIN {X 0,Y 281.95,Z 350.675,A -85,B 0,C 180,E1 -19230.634,E2 -19230.634} C_VEL
LIN {X 0,Y 277.58,Z 344.411,A -85,B 0,C 180,E1 -19233.194,E2 -19233.194} C_VEL
LIN {X 0,Y 274.763,Z 340.992,A -85,B 0,C 180,E1 -19235.025,E2 -19235.025} C_VEL
LIN {X 0,Y 273.953,Z 339.718,A -85,B 0,C 180,E1 -19235.618,E2 -19235.618} C_VEL
LIN {X 0,Y 271.192,Z 336.905,A -85,B 0,C 180,E1 -19237.682,E2 -19237.682} C_VEL
LIN {X 0,Y 269.716,Z 334.489,A -85,B 0,C 180,E1 -19239.006,E2 -19239.006} C_VEL
LIN {X 0,Y 266.931,Z 331.995,A -85,B 0,C 180,E1 -19241.707,E2 -19241.707} C_VEL
LIN {X 0,Y 265.314,Z 328.888,A -85,B 0,C 180,E1 -19243.903,E2 -19243.903} C_VEL
LIN {X 0,Y 261.742,Z 325.753,A -85,B 0,C 180,E1 -19252.285,E2 -19252.285} C_VEL
LIN {X 0,Y 261.681,Z 325.772,A -85,B 0,C 180,E1 -19254.607,E2 -19254.607} C_VEL
LIN {X 0,Y 262.804,Z 326.931,A -85,B 0,C 180,E1 -19259.235,E2 -19259.235} C_VEL
LIN {X 0,Y 265.709,Z 329.158,A -85,B 0,C 180,E1 -19264.051,E2 -19264.051} C_VEL
LIN {X 0,Y 267.4,Z 332.267,A -85,B 0,C 180,E1 -19266.225,E2 -19266.225} C_VEL
LIN {X 0,Y 270.167,Z 334.862,A -85,B 0,C 180,E1 -19268.822,E2 -19268.822} C_VEL
LIN {X 0,Y 272.196,Z 338.024,A -85,B 0,C 180,E1 -19270.555,E2 -19270.555} C_VEL
LIN {X 0,Y 274.358,Z 340.116,A -85,B 0,C 180,E1 -19272.107,E2 -19272.107} C_VEL
LIN {X 0,Y 276.93,Z 343.759,A -85,B 0,C 180,E1 -19273.858,E2 -19273.858} C_VEL
LIN {X 0,Y 278.437,Z 345.452,A -85,B 0,C 180,E1 -19274.77,E2 -19274.77} C_VEL
LIN {X 0,Y 282.391,Z 350.746,A -85,B 0,C 180,E1 -19277.017,E2 -19277.017} C_VEL
LIN {X 0,Y 285.954,Z 355.54,A -85,B 0,C 180,E1 -19278.837,E2 -19278.837} C_VEL
LIN {X 0,Y 291.164,Z 362.707,A -85,B 0,C 180,E1 -19281.228,E2 -19281.228} C_VEL
LIN {X 0,Y 298.628,Z 373.914,A -85,B 0,C 180,E1 -19284.266,E2 -19284.266} C_VEL
LIN {X 0,Y 305.259,Z 384.882,A -85,B 0,C 180,E1 -19286.677,E2 -19286.677} C_VEL
LIN {X 0,Y 307.886,Z 389.416,A -85,B 0,C 180,E1 -19287.569,E2 -19287.569} C_VEL
LIN {X 0,Y 300.506,Z 499.293,A -85,B 0,C 180,E1 -19290.079,E2 -19290.079} C_VEL
LIN {X 0,Y 298.337,Z 515.967,A -85,B 0,C 180,E1 -19290.66,E2 -19290.66} C_VEL
LIN {X 0,Y 295.684,Z 531.387,A -85,B 0,C 180,E1 -19291.445,E2 -19291.445} C_VEL
LIN {X 0,Y 292.32,Z 546.781,A -85,B 0,C 180,E1 -19292.467,E2 -19292.467} C_VEL
LIN {X 0,Y 288.804,Z 559.931,A -85,B 0,C 180,E1 -19293.543,E2 -19293.543} C_VEL
LIN {X 0,Y 284.369,Z 574.184,A -85,B 0,C 180,E1 -19294.994,E2 -19294.994} C_VEL
LIN {X 0,Y 279.252,Z 588.645,A -85,B 0,C 180,E1 -19296.821,E2 -19296.821} C_VEL
LIN {X 0,Y 274.018,Z 601.649,A -85,B 0,C 180,E1 -19298.825,E2 -19298.825} C_VEL
LIN {X 0,Y 269.381,Z 612.358,A -85,B 0,C 180,E1 -19300.835,E2 -19300.835} C_VEL
LIN {X 0,Y 264.646,Z 622.404,A -85,B 0,C 180,E1 -19303.088,E2 -19303.088} C_VEL
LIN {X 0,Y 259.593,Z 632.489,A -85,B 0,C 180,E1 -19305.802,E2 -19305.802} C_VEL
LIN {X 0,Y 254.626,Z 642.161,A -85,B 0,C 180,E1 -19309.04,E2 -19309.04} C_VEL
LIN {X 0,Y 250.902,Z 649.176,A -85,B 0,C 180,E1 -19311.958,E2 -19311.958} C_VEL
LIN {X 0,Y 247.167,Z 656.153,A -85,B 0,C 180,E1 -19315.549,E2 -19315.549} C_VEL
LIN {X 0,Y 244.517,Z 661.221,A -85,B 0,C 180,E1 -19318.844,E2 -19318.844} C_VEL
LIN {X 0,Y 242.428,Z 665.294,A -85,B 0,C 180,E1 -19322.365,E2 -19322.365} C_VEL
LIN {X 0,Y 241,Z 668.263,A -85,B 0,C 180,E1 -19325.904,E2 -19325.904} C_VEL
LIN {X 0,Y 240.111,Z 670.19,A -85,B 0,C 180,E1 -19329.496,E2 -19329.496} C_VEL
LIN {X 0,Y 239.651,Z 670.992,A -85,B 0,C 180,E1 -19332.947,E2 -19332.947} C_VEL
LIN {X 0,Y 239.576,Z 670.876,A -85,B 0,C 180,E1 -19336.427,E2 -19336.427} C_VEL
LIN {X 0,Y 239.576,Z 669.702,A -85,B 0,C 180,E1 -19339.862,E2 -19339.862} C_VEL
LIN {X 0,Y 239.901,Z 667.632,A -85,B 0,C 180,E1 -19343.27,E2 -19343.27} C_VEL
LIN {X 0,Y 240.402,Z 664.476,A -85,B 0,C 180,E1 -19346.648,E2 -19346.648} C_VEL
LIN {X 0,Y 241.238,Z 660.367,A -85,B 0,C 180,E1 -19350,E2 -19350} C_VEL
LIN {X 0,Y 242.48,Z 655.115,A -85,B 0,C 180,E1 -19353.323,E2 -19353.323} C_VEL
LIN {X 0,Y 244.371,Z 648.687,A -85,B 0,C 180,E1 -19356.606,E2 -19356.606} C_VEL
LIN {X 0,Y 246.854,Z 640.989,A -85,B 0,C 180,E1 -19359.835,E2 -19359.835} C_VEL
LIN {X 0,Y 250.068,Z 631.713,A -85,B 0,C 180,E1 -19362.993,E2 -19362.993} C_VEL
LIN {X 0,Y 253.259,Z 622.165,A -85,B 0,C 180,E1 -19365.698,E2 -19365.698} C_VEL
LIN {X 0,Y 256.88,Z 611.065,A -85,B 0,C 180,E1 -19368.338,E2 -19368.338} C_VEL
LIN {X 0,Y 260.568,Z 599.031,A -85,B 0,C 180,E1 -19370.732,E2 -19370.732} C_VEL
LIN {X 0,Y 264.3,Z 585.874,A -85,B 0,C 180,E1 -19372.885,E2 -19372.885} C_VEL
LIN {X 0,Y 268.119,Z 571.531,A -85,B 0,C 180,E1 -19374.796,E2 -19374.796} C_VEL
LIN {X 0,Y 271.346,Z 557.541,A -85,B 0,C 180,E1 -19376.33,E2 -19376.33} C_VEL
LIN {X 0,Y 274.232,Z 542.545,A -85,B 0,C 180,E1 -19377.678,E2 -19377.678} C_VEL
LIN {X 0,Y 277.127,Z 525.745,A -85,B 0,C 180,E1 -19378.806,E2 -19378.806} C_VEL
LIN {X 0,Y 279.141,Z 509.608,A -85,B 0,C 180,E1 -19379.61,E2 -19379.61} C_VEL
LIN {X 0,Y 280.607,Z 493.196,A -85,B 0,C 180,E1 -19380.164,E2 -19380.164} C_VEL
LIN {X 0,Y 286.835,Z 375.487,A -85,B 0,C 180,E1 -19382.982,E2 -19382.982} C_VEL
LIN {X 0,Y 282.213,Z 366.179,A -85,B 0,C 180,E1 -19384.127,E2 -19384.127} C_VEL
LIN {X 0,Y 272.695,Z 349.419,A -85,B 0,C 180,E1 -19386.589,E2 -19386.589} C_VEL
LIN {X 0,Y 264.188,Z 335.895,A -85,B 0,C 180,E1 -19388.971,E2 -19388.971} C_VEL
LIN {X 0,Y 257.527,Z 326.412,A -85,B 0,C 180,E1 -19390.982,E2 -19390.982} C_VEL
LIN {X 0,Y 254.775,Z 322.671,A -85,B 0,C 180,E1 -19391.857,E2 -19391.857} C_VEL
LIN {X 0,Y 252.017,Z 318.854,A -85,B 0,C 180,E1 -19392.77,E2 -19392.77} C_VEL
LIN {X 0,Y 249.486,Z 315.303,A -85,B 0,C 180,E1 -19393.645,E2 -19393.645} C_VEL
LIN {X 0,Y 246.573,Z 311.9,A -85,B 0,C 180,E1 -19394.663,E2 -19394.663} C_VEL
LIN {X 0,Y 245.345,Z 309.857,A -85,B 0,C 180,E1 -19395.136,E2 -19395.136} C_VEL
LIN {X 0,Y 243.198,Z 307.935,A -85,B 0,C 180,E1 -19395.906,E2 -19395.906} C_VEL
LIN {X 0,Y 242.043,Z 305.479,A -85,B 0,C 180,E1 -19396.403,E2 -19396.403} C_VEL
LIN {X 0,Y 241.893,Z 304.647,A -85,B 0,C 180,E1 -19396.536,E2 -19396.536} C_VEL
LIN {X 0,Y 241.932,Z 304.634,A -85,B 0,C 180,E1 -19400.275,E2 -19400.275} C_VEL
LIN {X 0,Y 241.975,Z 304.59,A -85,B 0,C 180,E1 -19404.486,E2 -19404.486} C_VEL
LIN {X 0,Y 241.951,Z 304.659,A -85,B 0,C 180,E1 -19408.475,E2 -19408.475} C_VEL
LIN {X 0,Y 241.962,Z 304.647,A -85,B 0,C 180,E1 -19412.306,E2 -19412.306} C_VEL
LIN {X 0,Y 242.006,Z 304.63,A -85,B 0,C 180,E1 -19416.306,E2 -19416.306} C_VEL
LIN {X 0,Y 241.298,Z 304.728,A -85,B 0,C 180,E1 -19417.695,E2 -19417.695} C_VEL
LIN {X 0,Y 238.472,Z 305.089,A -85,B 0,C 180,E1 -19419.963,E2 -19419.963} C_VEL
LIN {X 0,Y 236.114,Z 305.371,A -85,B 0,C 180,E1 -19421.81,E2 -19421.81} C_VEL
LIN {X 0,Y 235.125,Z 305.491,A -85,B 0,C 180,E1 -19423.242,E2 -19423.242} C_VEL
LIN {X 0,Y 235.054,Z 305.504,A -85,B 0,C 180,E1 -19423.727,E2 -19423.727} C_VEL
LIN {X 0,Y 235.111,Z 305.487,A -85,B 0,C 180,E1 -19427.921,E2 -19427.921} C_VEL
LIN {X 0,Y 235.326,Z 305.485,A -85,B 0,C 180,E1 -19431.411,E2 -19431.411} C_VEL
LIN {X 0,Y 235.365,Z 305.46,A -85,B 0,C 180,E1 -19433.139,E2 -19433.139} C_VEL
LIN {X 0,Y 235.591,Z 305.445,A -85,B 0,C 180,E1 -19438.29,E2 -19438.29} C_VEL
LIN {X 0,Y 235.595,Z 305.433,A -85,B 0,C 180,E1 -19441.709,E2 -19441.709} C_VEL
LIN {X 0,Y 235.371,Z 305.442,A -85,B 0,C 180,E1 -19446.859,E2 -19446.859} C_VEL
LIN {X 0,Y 235.214,Z 305.499,A -85,B 0,C 180,E1 -19450.327,E2 -19450.327} C_VEL
LIN {X 0,Y 235.093,Z 305.508,A -85,B 0,C 180,E1 -19455.607,E2 -19455.607} C_VEL
LIN {X 0,Y 234.999,Z 305.521,A -85,B 0,C 180,E1 -19459.205,E2 -19459.205} C_VEL
LIN {X 0,Y 234.96,Z 305.528,A -85,B 0,C 180,E1 -19462.882,E2 -19462.882} C_VEL
LIN {X 0,Y 234.968,Z 305.534,A -85,B 0,C 180,E1 -19466.657,E2 -19466.657} C_VEL
LIN {X 0,Y 234.968,Z 305.526,A -85,B 0,C 180,E1 -19467.74,E2 -19467.74} C_VEL
LIN {X 0,Y 235.856,Z 308.191,A -85,B 0,C 180,E1 -19468.231,E2 -19468.231} C_VEL
LIN {X 0,Y 237.789,Z 310.331,A -85,B 0,C 180,E1 -19469.03,E2 -19469.03} C_VEL
LIN {X 0,Y 239.023,Z 311.362,A -85,B 0,C 180,E1 -19469.508,E2 -19469.508} C_VEL
LIN {X 0,Y 240.982,Z 314.546,A -85,B 0,C 180,E1 -19470.324,E2 -19470.324} C_VEL
LIN {X 0,Y 242.978,Z 316.686,A -85,B 0,C 180,E1 -19471.071,E2 -19471.071} C_VEL
LIN {X 0,Y 245.465,Z 320.104,A -85,B 0,C 180,E1 -19472.004,E2 -19472.004} C_VEL
LIN {X 0,Y 247.032,Z 322.106,A -85,B 0,C 180,E1 -19472.566,E2 -19472.566} C_VEL
LIN {X 0,Y 250.857,Z 327.296,A -85,B 0,C 180,E1 -19473.895,E2 -19473.895} C_VEL
LIN {X 0,Y 255.67,Z 334.105,A -85,B 0,C 180,E1 -19475.483,E2 -19475.483} C_VEL
LIN {X 0,Y 262.111,Z 345.249,A -85,B 0,C 180,E1 -19477.528,E2 -19477.528} C_VEL
LIN {X 0,Y 269.379,Z 358.706,A -85,B 0,C 180,E1 -19479.67,E2 -19479.67} C_VEL
LIN {X 0,Y 276.118,Z 372.722,A -85,B 0,C 180,E1 -19481.556,E2 -19481.556} C_VEL
LIN {X 0,Y 281.211,Z 384.398,A -85,B 0,C 180,E1 -19482.923,E2 -19482.923} C_VEL
LIN {X 0,Y 274.401,Z 509.595,A -85,B 0,C 180,E1 -19485.986,E2 -19485.986} C_VEL
LIN {X 0,Y 272.673,Z 525.957,A -85,B 0,C 180,E1 -19486.603,E2 -19486.603} C_VEL
LIN {X 0,Y 270.268,Z 542.098,A -85,B 0,C 180,E1 -19487.461,E2 -19487.461} C_VEL
LIN {X 0,Y 267.644,Z 556.495,A -85,B 0,C 180,E1 -19488.468,E2 -19488.468} C_VEL
LIN {X 0,Y 264.274,Z 571.79,A -85,B 0,C 180,E1 -19489.842,E2 -19489.842} C_VEL
LIN {X 0,Y 260.47,Z 586.479,A -85,B 0,C 180,E1 -19491.487,E2 -19491.487} C_VEL
LIN {X 0,Y 256.576,Z 600.456,A -85,B 0,C 180,E1 -19493.433,E2 -19493.433} C_VEL
LIN {X 0,Y 253.137,Z 611.765,A -85,B 0,C 180,E1 -19495.309,E2 -19495.309} C_VEL
LIN {X 0,Y 248.824,Z 624.786,A -85,B 0,C 180,E1 -19497.923,E2 -19497.923} C_VEL
LIN {X 0,Y 245.459,Z 634.962,A -85,B 0,C 180,E1 -19500.403,E2 -19500.403} C_VEL
LIN {X 0,Y 242.031,Z 644.882,A -85,B 0,C 180,E1 -19503.251,E2 -19503.251} C_VEL
LIN {X 0,Y 238.909,Z 654.47,A -85,B 0,C 180,E1 -19506.601,E2 -19506.601} C_VEL
LIN {X 0,Y 236.447,Z 662.401,A -85,B 0,C 180,E1 -19510.012,E2 -19510.012} C_VEL
LIN {X 0,Y 234.721,Z 668.791,A -85,B 0,C 180,E1 -19513.361,E2 -19513.361} C_VEL
LIN {X 0,Y 233.564,Z 674.346,A -85,B 0,C 180,E1 -19516.958,E2 -19516.958} C_VEL
LIN {X 0,Y 232.818,Z 679.376,A -85,B 0,C 180,E1 -19521.319,E2 -19521.319} C_VEL
LIN {X 0,Y 232.751,Z 682.38,A -85,B 0,C 180,E1 -19525.159,E2 -19525.159} C_VEL
LIN {X 0,Y 232.752,Z 683.971,A -85,B 0,C 180,E1 -19528.27,E2 -19528.27} C_VEL
LIN {X 0,Y 232.821,Z 684.451,A -85,B 0,C 180,E1 -19530,E2 -19530} C_VEL
LIN {X 0,Y 232.65,Z 684.738,A -85,B 0,C 180,E1 -19533.464,E2 -19533.464} C_VEL
LIN {X 0,Y 232.676,Z 684.054,A -85,B 0,C 180,E1 -19536.94,E2 -19536.94} C_VEL
LIN {X 0,Y 233.039,Z 682.433,A -85,B 0,C 180,E1 -19540.425,E2 -19540.425} C_VEL
LIN {X 0,Y 233.966,Z 679.826,A -85,B 0,C 180,E1 -19543.905,E2 -19543.905} C_VEL
LIN {X 0,Y 235.933,Z 675.17,A -85,B 0,C 180,E1 -19548.227,E2 -19548.227} C_VEL
LIN {X 0,Y 238.342,Z 670.292,A -85,B 0,C 180,E1 -19551.629,E2 -19551.629} C_VEL
LIN {X 0,Y 241.423,Z 664.243,A -85,B 0,C 180,E1 -19554.968,E2 -19554.968} C_VEL
LIN {X 0,Y 245.289,Z 656.951,A -85,B 0,C 180,E1 -19558.214,E2 -19558.214} C_VEL
LIN {X 0,Y 249.946,Z 648.302,A -85,B 0,C 180,E1 -19561.345,E2 -19561.345} C_VEL
LIN {X 0,Y 254.975,Z 638.546,A -85,B 0,C 180,E1 -19564.219,E2 -19564.219} C_VEL
LIN {X 0,Y 260.525,Z 627.372,A -85,B 0,C 180,E1 -19566.886,E2 -19566.886} C_VEL
LIN {X 0,Y 266.317,Z 614.945,A -85,B 0,C 180,E1 -19569.298,E2 -19569.298} C_VEL
LIN {X 0,Y 271.8,Z 601.975,A -85,B 0,C 180,E1 -19571.36,E2 -19571.36} C_VEL
LIN {X 0,Y 277.311,Z 587.706,A -85,B 0,C 180,E1 -19573.179,E2 -19573.179} C_VEL
LIN {X 0,Y 282.371,Z 572.867,A -85,B 0,C 180,E1 -19574.678,E2 -19574.678} C_VEL
LIN {X 0,Y 286.456,Z 558.434,A -85,B 0,C 180,E1 -19575.859,E2 -19575.859} C_VEL
LIN {X 0,Y 290.218,Z 542.867,A -85,B 0,C 180,E1 -19576.846,E2 -19576.846} C_VEL
LIN {X 0,Y 293.269,Z 527.101,A -85,B 0,C 180,E1 -19577.596,E2 -19577.596} C_VEL
LIN {X 0,Y 295.585,Z 510.372,A -85,B 0,C 180,E1 -19578.162,E2 -19578.162} C_VEL
LIN {X 0,Y 300.304,Z 442.764,A -85,B 0,C 180,E1 -19579.734,E2 -19579.734} C_VEL
LIN {X 0,Y 303.267,Z 398.342,A -85,B 0,C 180,E1 -19580.76,E2 -19580.76} C_VEL
LIN {X 0,Y 297.38,Z 386.472,A -85,B 0,C 180,E1 -19582.997,E2 -19582.997} C_VEL
LIN {X 0,Y 291.764,Z 376.168,A -85,B 0,C 180,E1 -19585.328,E2 -19585.328} C_VEL
LIN {X 0,Y 285.71,Z 365.882,A -85,B 0,C 180,E1 -19588.124,E2 -19588.124} C_VEL
LIN {X 0,Y 282.446,Z 360.896,A -85,B 0,C 180,E1 -19589.786,E2 -19589.786} C_VEL
LIN {X 0,Y 279.75,Z 356.686,A -85,B 0,C 180,E1 -19591.28,E2 -19591.28} C_VEL
LIN {X 0,Y 275.748,Z 350.873,A -85,B 0,C 180,E1 -19593.716,E2 -19593.716} C_VEL
LIN {X 0,Y 272.901,Z 347.133,A -85,B 0,C 180,E1 -19595.667,E2 -19595.667} C_VEL
LIN {X 0,Y 272.18,Z 346.246,A -85,B 0,C 180,E1 -19596.196,E2 -19596.196} C_VEL
LIN {X 0,Y 269.368,Z 342.98,A -85,B 0,C 180,E1 -19598.437,E2 -19598.437} C_VEL
LIN {X 0,Y 268.403,Z 341.32,A -85,B 0,C 180,E1 -19599.35,E2 -19599.35} C_VEL
LIN {X 0,Y 265.671,Z 338.722,A -85,B 0,C 180,E1 -19602.114,E2 -19602.114} C_VEL
LIN {X 0,Y 264.309,Z 335.893,A -85,B 0,C 180,E1 -19604.05,E2 -19604.05} C_VEL
LIN {X 0,Y 260.87,Z 332.795,A -85,B 0,C 180,E1 -19612.259,E2 -19612.259} C_VEL
LIN {X 0,Y 260.803,Z 332.82,A -85,B 0,C 180,E1 -19614.589,E2 -19614.589} C_VEL
LIN {X 0,Y 261.919,Z 333.993,A -85,B 0,C 180,E1 -19619.232,E2 -19619.232} C_VEL
LIN {X 0,Y 264.616,Z 336.219,A -85,B 0,C 180,E1 -19623.818,E2 -19623.818} C_VEL
LIN {X 0,Y 266.336,Z 339.252,A -85,B 0,C 180,E1 -19626.06,E2 -19626.06} C_VEL
LIN {X 0,Y 268.686,Z 341.433,A -85,B 0,C 180,E1 -19628.332,E2 -19628.332} C_VEL
LIN {X 0,Y 270.872,Z 344.86,A -85,B 0,C 180,E1 -19630.26,E2 -19630.26} C_VEL
LIN {X 0,Y 272.899,Z 346.938,A -85,B 0,C 180,E1 -19631.761,E2 -19631.761} C_VEL
LIN {X 0,Y 275.544,Z 350.632,A -85,B 0,C 180,E1 -19633.6,E2 -19633.6} C_VEL
LIN {X 0,Y 276.965,Z 352.408,A -85,B 0,C 180,E1 -19634.489,E2 -19634.489} C_VEL
LIN {X 0,Y 280.352,Z 356.99,A -85,B 0,C 180,E1 -19636.468,E2 -19636.468} C_VEL
LIN {X 0,Y 284.165,Z 362.29,A -85,B 0,C 180,E1 -19638.48,E2 -19638.48} C_VEL
LIN {X 0,Y 289.196,Z 369.44,A -85,B 0,C 180,E1 -19640.856,E2 -19640.856} C_VEL
LIN {X 0,Y 295.661,Z 379.314,A -85,B 0,C 180,E1 -19643.574,E2 -19643.574} C_VEL
LIN {X 0,Y 302.241,Z 390.399,A -85,B 0,C 180,E1 -19646.064,E2 -19646.064} C_VEL
LIN {X 0,Y 303.578,Z 392.792,A -85,B 0,C 180,E1 -19646.541,E2 -19646.541} C_VEL
LIN {X 0,Y 296.258,Z 498.853,A -85,B 0,C 180,E1 -19648.982,E2 -19648.982} C_VEL
LIN {X 0,Y 294.076,Z 515.24,A -85,B 0,C 180,E1 -19649.534,E2 -19649.534} C_VEL
LIN {X 0,Y 291.406,Z 530.66,A -85,B 0,C 180,E1 -19650.307,E2 -19650.307} C_VEL
LIN {X 0,Y 287.959,Z 546.21,A -85,B 0,C 180,E1 -19651.326,E2 -19651.326} C_VEL
LIN {X 0,Y 284.72,Z 558.072,A -85,B 0,C 180,E1 -19652.282,E2 -19652.282} C_VEL
LIN {X 0,Y 279.991,Z 573.185,A -85,B 0,C 180,E1 -19653.791,E2 -19653.791} C_VEL
LIN {X 0,Y 275.08,Z 586.734,A -85,B 0,C 180,E1 -19655.454,E2 -19655.454} C_VEL
LIN {X 0,Y 269.826,Z 599.657,A -85,B 0,C 180,E1 -19657.4,E2 -19657.4} C_VEL
LIN {X 0,Y 263.899,Z 612.8,A -85,B 0,C 180,E1 -19659.853,E2 -19659.853} C_VEL
LIN {X 0,Y 258.726,Z 623.273,A -85,B 0,C 180,E1 -19662.25,E2 -19662.25} C_VEL
LIN {X 0,Y 253.483,Z 633.244,A -85,B 0,C 180,E1 -19665.008,E2 -19665.008} C_VEL
LIN {X 0,Y 248.907,Z 641.741,A -85,B 0,C 180,E1 -19667.887,E2 -19667.887} C_VEL
LIN {X 0,Y 244.941,Z 648.846,A -85,B 0,C 180,E1 -19670.858,E2 -19670.858} C_VEL
LIN {X 0,Y 241.118,Z 655.629,A -85,B 0,C 180,E1 -19674.341,E2 -19674.341} C_VEL
LIN {X 0,Y 238.061,Z 661.083,A -85,B 0,C 180,E1 -19677.9,E2 -19677.9} C_VEL
LIN {X 0,Y 235.743,Z 665.237,A -85,B 0,C 180,E1 -19681.51,E2 -19681.51} C_VEL
LIN {X 0,Y 234.168,Z 668.308,A -85,B 0,C 180,E1 -19685.154,E2 -19685.154} C_VEL
LIN {X 0,Y 233.061,Z 670.437,A -85,B 0,C 180,E1 -19689.2,E2 -19689.2} C_VEL
LIN {X 0,Y 232.603,Z 671.182,A -85,B 0,C 180,E1 -19692.413,E2 -19692.413} C_VEL
LIN {X 0,Y 232.485,Z 671.111,A -85,B 0,C 180,E1 -19696.005,E2 -19696.005} C_VEL
LIN {X 0,Y 232.453,Z 670.03,A -85,B 0,C 180,E1 -19699.548,E2 -19699.548} C_VEL
LIN {X 0,Y 232.771,Z 668.013,A -85,B 0,C 180,E1 -19703.063,E2 -19703.063} C_VEL
LIN {X 0,Y 233.308,Z 664.941,A -85,B 0,C 180,E1 -19706.546,E2 -19706.546} C_VEL
LIN {X 0,Y 234.146,Z 660.925,A -85,B 0,C 180,E1 -19710,E2 -19710} C_VEL
LIN {X 0,Y 235.855,Z 654.31,A -85,B 0,C 180,E1 -19714.272,E2 -19714.272} C_VEL
LIN {X 0,Y 237.903,Z 647.624,A -85,B 0,C 180,E1 -19717.639,E2 -19717.639} C_VEL
LIN {X 0,Y 240.639,Z 639.626,A -85,B 0,C 180,E1 -19720.943,E2 -19720.943} C_VEL
LIN {X 0,Y 244.093,Z 630.101,A -85,B 0,C 180,E1 -19724.166,E2 -19724.166} C_VEL
LIN {X 0,Y 247.528,Z 620.285,A -85,B 0,C 180,E1 -19726.919,E2 -19726.919} C_VEL
LIN {X 0,Y 251.357,Z 608.775,A -85,B 0,C 180,E1 -19729.604,E2 -19729.604} C_VEL
LIN {X 0,Y 255.273,Z 596.242,A -85,B 0,C 180,E1 -19732.031,E2 -19732.031} C_VEL
LIN {X 0,Y 259.241,Z 582.591,A -85,B 0,C 180,E1 -19734.207,E2 -19734.207} C_VEL
LIN {X 0,Y 262.884,Z 569.115,A -85,B 0,C 180,E1 -19735.962,E2 -19735.962} C_VEL
LIN {X 0,Y 266.196,Z 554.517,A -85,B 0,C 180,E1 -19737.518,E2 -19737.518} C_VEL
LIN {X 0,Y 269.088,Z 539.695,A -85,B 0,C 180,E1 -19738.786,E2 -19738.786} C_VEL
LIN {X 0,Y 271.838,Z 523.374,A -85,B 0,C 180,E1 -19739.847,E2 -19739.847} C_VEL
LIN {X 0,Y 273.85,Z 507.509,A -85,B 0,C 180,E1 -19740.615,E2 -19740.615} C_VEL
LIN {X 0,Y 275.335,Z 489.776,A -85,B 0,C 180,E1 -19741.177,E2 -19741.177} C_VEL
LIN {X 0,Y 281.378,Z 378.241,A -85,B 0,C 180,E1 -19743.87,E2 -19743.87} C_VEL
LIN {X 0,Y 280.922,Z 376.713,A -85,B 0,C 180,E1 -19744.006,E2 -19744.006} C_VEL
LIN {X 0,Y 273.404,Z 362.644,A -85,B 0,C 180,E1 -19745.961,E2 -19745.961} C_VEL
LIN {X 0,Y 265.988,Z 349.953,A -85,B 0,C 180,E1 -19748.013,E2 -19748.013} C_VEL
LIN {X 0,Y 259.11,Z 339.175,A -85,B 0,C 180,E1 -19750.054,E2 -19750.054} C_VEL
LIN {X 0,Y 252.256,Z 329.203,A -85,B 0,C 180,E1 -19752.248,E2 -19752.248} C_VEL
LIN {X 0,Y 248.07,Z 323.685,A -85,B 0,C 180,E1 -19753.669,E2 -19753.669} C_VEL
LIN {X 0,Y 245.631,Z 320.305,A -85,B 0,C 180,E1 -19754.55,E2 -19754.55} C_VEL
LIN {X 0,Y 242.982,Z 316.771,A -85,B 0,C 180,E1 -19755.54,E2 -19755.54} C_VEL
LIN {X 0,Y 241.968,Z 315.607,A -85,B 0,C 180,E1 -19755.922,E2 -19755.922} C_VEL
LIN {X 0,Y 239.528,Z 312.654,A -85,B 0,C 180,E1 -19756.872,E2 -19756.872} C_VEL
LIN {X 0,Y 238.759,Z 311.009,A -85,B 0,C 180,E1 -19757.216,E2 -19757.216} C_VEL
LIN {X 0,Y 236.324,Z 309.057,A -85,B 0,C 180,E1 -19758.167,E2 -19758.167} C_VEL
LIN {X 0,Y 235.084,Z 306.622,A -85,B 0,C 180,E1 -19758.746,E2 -19758.746} C_VEL
LIN {X 0,Y 234.866,Z 305.543,A -85,B 0,C 180,E1 -19758.898,E2 -19758.898} C_VEL
LIN {X 0,Y 234.92,Z 305.486,A -85,B 0,C 180,E1 -19761.078,E2 -19761.078} C_VEL
LIN {X 0,Y 234.903,Z 305.481,A -85,B 0,C 180,E1 -19765.356,E2 -19765.356} C_VEL
LIN {X 0,Y 234.954,Z 305.524,A -85,B 0,C 180,E1 -19767.423,E2 -19767.423} C_VEL
LIN {X 0,Y 234.897,Z 305.518,A -85,B 0,C 180,E1 -19771.398,E2 -19771.398} C_VEL
LIN {X 0,Y 234.954,Z 305.513,A -85,B 0,C 180,E1 -19775.242,E2 -19775.242} C_VEL
LIN {X 0,Y 234.991,Z 305.526,A -85,B 0,C 180,E1 -19778.967,E2 -19778.967} C_VEL
LIN {X 0,Y 235.054,Z 305.504,A -85,B 0,C 180,E1 -19783.727,E2 -19783.727} C_VEL
LIN {X 0,Y 234.437,Z 305.599,A -85,B 0,C 180,E1 -19785.157,E2 -19785.157} C_VEL
LIN {X 0,Y 231.702,Z 305.957,A -85,B 0,C 180,E1 -19787.493,E2 -19787.493} C_VEL
LIN {X 0,Y 228.57,Z 306.336,A -85,B 0,C 180,E1 -19790.375,E2 -19790.375} C_VEL
LIN {X 0,Y 228.258,Z 306.362,A -85,B 0,C 180,E1 -19791.371,E2 -19791.371} C_VEL
LIN {X 0,Y 228.163,Z 306.352,A -85,B 0,C 180,E1 -19794.697,E2 -19794.697} C_VEL
LIN {X 0,Y 228.55,Z 306.322,A -85,B 0,C 180,E1 -19798.237,E2 -19798.237} C_VEL
LIN {X 0,Y 228.554,Z 306.31,A -85,B 0,C 180,E1 -19801.761,E2 -19801.761} C_VEL
LIN {X 0,Y 228.322,Z 306.319,A -85,B 0,C 180,E1 -19807.072,E2 -19807.072} C_VEL
LIN {X 0,Y 228.145,Z 306.38,A -85,B 0,C 180,E1 -19810.65,E2 -19810.65} C_VEL
LIN {X 0,Y 228.05,Z 306.393,A -85,B 0,C 180,E1 -19814.272,E2 -19814.272} C_VEL
LIN {X 0,Y 227.997,Z 306.399,A -85,B 0,C 180,E1 -19817.953,E2 -19817.953} C_VEL
LIN {X 0,Y 227.929,Z 306.402,A -85,B 0,C 180,E1 -19822.329,E2 -19822.329} C_VEL
LIN {X 0,Y 227.968,Z 306.594,A -85,B 0,C 180,E1 -19825.08,E2 -19825.08} C_VEL
LIN {X 0,Y 228.805,Z 309.044,A -85,B 0,C 180,E1 -19825.573,E2 -19825.573} C_VEL
LIN {X 0,Y 230.898,Z 311.345,A -85,B 0,C 180,E1 -19826.544,E2 -19826.544} C_VEL
LIN {X 0,Y 232.133,Z 312.219,A -85,B 0,C 180,E1 -19827.069,E2 -19827.069} C_VEL
LIN {X 0,Y 233.965,Z 315.34,A -85,B 0,C 180,E1 -19827.93,E2 -19827.93} C_VEL
LIN {X 0,Y 236.299,Z 317.72,A -85,B 0,C 180,E1 -19828.899,E2 -19828.899} C_VEL
LIN {X 0,Y 238.826,Z 321.245,A -85,B 0,C 180,E1 -19829.95,E2 -19829.95} C_VEL
LIN {X 0,Y 240.153,Z 322.855,A -85,B 0,C 180,E1 -19830.47,E2 -19830.47} C_VEL
LIN {X 0,Y 244.308,Z 328.438,A -85,B 0,C 180,E1 -19832.05,E2 -19832.05} C_VEL
LIN {X 0,Y 249.703,Z 335.743,A -85,B 0,C 180,E1 -19833.952,E2 -19833.952} C_VEL
LIN {X 0,Y 253.601,Z 342.048,A -85,B 0,C 180,E1 -19835.284,E2 -19835.284} C_VEL
LIN {X 0,Y 259.586,Z 352.576,A -85,B 0,C 180,E1 -19837.223,E2 -19837.223} C_VEL
LIN {X 0,Y 266.118,Z 365.16,A -85,B 0,C 180,E1 -19839.21,E2 -19839.21} C_VEL
LIN {X 0,Y 272.105,Z 378.052,A -85,B 0,C 180,E1 -19840.948,E2 -19840.948} C_VEL
LIN {X 0,Y 275.806,Z 386.518,A -85,B 0,C 180,E1 -19841.982,E2 -19841.982} C_VEL
LIN {X 0,Y 268.876,Z 510.091,A -85,B 0,C 180,E1 -19845.051,E2 -19845.051} C_VEL
LIN {X 0,Y 267.023,Z 526.904,A -85,B 0,C 180,E1 -19845.709,E2 -19845.709} C_VEL
LIN {X 0,Y 264.533,Z 542.705,A -85,B 0,C 180,E1 -19846.573,E2 -19846.573} C_VEL
LIN {X 0,Y 261.631,Z 557.928,A -85,B 0,C 180,E1 -19847.683,E2 -19847.683} C_VEL
LIN {X 0,Y 258.37,Z 572.138,A -85,B 0,C 180,E1 -19848.987,E2 -19848.987} C_VEL
LIN {X 0,Y 254.442,Z 586.742,A -85,B 0,C 180,E1 -19850.658,E2 -19850.658} C_VEL
LIN {X 0,Y 250.425,Z 600.617,A -85,B 0,C 180,E1 -19852.635,E2 -19852.635} C_VEL
LIN {X 0,Y 246.554,Z 612.893,A -85,B 0,C 180,E1 -19854.745,E2 -19854.745} C_VEL
LIN {X 0,Y 242.384,Z 624.937,A -85,B 0,C 180,E1 -19857.23,E2 -19857.23} C_VEL
LIN {X 0,Y 238.632,Z 635.758,A -85,B 0,C 180,E1 -19859.956,E2 -19859.956} C_VEL
LIN {X 0,Y 235.118,Z 645.512,A -85,B 0,C 180,E1 -19862.881,E2 -19862.881} C_VEL
LIN {X 0,Y 231.923,Z 654.972,A -85,B 0,C 180,E1 -19866.327,E2 -19866.327} C_VEL
LIN {X 0,Y 229.114,Z 663.713,A -85,B 0,C 180,E1 -19870.28,E2 -19870.28} C_VEL
LIN {X 0,Y 227.424,Z 669.985,A -85,B 0,C 180,E1 -19873.852,E2 -19873.852} C_VEL
LIN {X 0,Y 226.299,Z 675.058,A -85,B 0,C 180,E1 -19877.444,E2 -19877.444} C_VEL
LIN {X 0,Y 225.736,Z 679.017,A -85,B 0,C 180,E1 -19881.045,E2 -19881.045} C_VEL
LIN {X 0,Y 225.662,Z 682.244,A -85,B 0,C 180,E1 -19885.267,E2 -19885.267} C_VEL
LIN {X 0,Y 225.666,Z 683.702,A -85,B 0,C 180,E1 -19888.216,E2 -19888.216} C_VEL
LIN {X 0,Y 225.732,Z 684.204,A -85,B 0,C 180,E1 -19890,E2 -19890} C_VEL
LIN {X 0,Y 225.568,Z 684.544,A -85,B 0,C 180,E1 -19893.573,E2 -19893.573} C_VEL
LIN {X 0,Y 225.59,Z 683.884,A -85,B 0,C 180,E1 -19897.159,E2 -19897.159} C_VEL
LIN {X 0,Y 226.006,Z 682.316,A -85,B 0,C 180,E1 -19900.753,E2 -19900.753} C_VEL
LIN {X 0,Y 227.016,Z 679.737,A -85,B 0,C 180,E1 -19904.34,E2 -19904.34} C_VEL
LIN {X 0,Y 228.595,Z 676.216,A -85,B 0,C 180,E1 -19907.905,E2 -19907.905} C_VEL
LIN {X 0,Y 231.662,Z 670.327,A -85,B 0,C 180,E1 -19912.285,E2 -19912.285} C_VEL
LIN {X 0,Y 234.914,Z 664.31,A -85,B 0,C 180,E1 -19915.709,E2 -19915.709} C_VEL
LIN {X 0,Y 239.018,Z 657.087,A -85,B 0,C 180,E1 -19919.023,E2 -19919.023} C_VEL
LIN {X 0,Y 243.853,Z 648.516,A -85,B 0,C 180,E1 -19922.221,E2 -19922.221} C_VEL
LIN {X 0,Y 249.523,Z 638.048,A -85,B 0,C 180,E1 -19925.356,E2 -19925.356} C_VEL
LIN {X 0,Y 255.667,Z 626.131,A -85,B 0,C 180,E1 -19928.207,E2 -19928.207} C_VEL
LIN {X 0,Y 261.79,Z 613.496,A -85,B 0,C 180,E1 -19930.618,E2 -19930.618} C_VEL
LIN {X 0,Y 266.913,Z 601.635,A -85,B 0,C 180,E1 -19932.503,E2 -19932.503} C_VEL
LIN {X 0,Y 272.225,Z 588.484,A -85,B 0,C 180,E1 -19934.192,E2 -19934.192} C_VEL
LIN {X 0,Y 277.423,Z 573.771,A -85,B 0,C 180,E1 -19935.698,E2 -19935.698} C_VEL
LIN {X 0,Y 281.623,Z 559.619,A -85,B 0,C 180,E1 -19936.882,E2 -19936.882} C_VEL
LIN {X 0,Y 285.48,Z 544.488,A -85,B 0,C 180,E1 -19937.87,E2 -19937.87} C_VEL
LIN {X 0,Y 288.738,Z 528.516,A -85,B 0,C 180,E1 -19938.656,E2 -19938.656} C_VEL
LIN {X 0,Y 291.235,Z 511.437,A -85,B 0,C 180,E1 -19939.243,E2 -19939.243} C_VEL
LIN {X 0,Y 293.431,Z 483.257,A -85,B 0,C 180,E1 -19939.931,E2 -19939.931} C_VEL
LIN {X 0,Y 299.128,Z 401.496,A -85,B 0,C 180,E1 -19941.805,E2 -19941.805} C_VEL
LIN {X 0,Y 293.031,Z 389.126,A -85,B 0,C 180,E1 -19944.268,E2 -19944.268} C_VEL
LIN {X 0,Y 287.973,Z 379.903,A -85,B 0,C 180,E1 -19946.496,E2 -19946.496} C_VEL
LIN {X 0,Y 283.163,Z 371.537,A -85,B 0,C 180,E1 -19948.85,E2 -19948.85} C_VEL
LIN {X 0,Y 280.495,Z 367.294,A -85,B 0,C 180,E1 -19950.266,E2 -19950.266} C_VEL
LIN {X 0,Y 277.629,Z 362.776,A -85,B 0,C 180,E1 -19951.912,E2 -19951.912} C_VEL
LIN {X 0,Y 274.188,Z 357.564,A -85,B 0,C 180,E1 -19954.088,E2 -19954.088} C_VEL
LIN {X 0,Y 271.241,Z 353.595,A -85,B 0,C 180,E1 -19956.182,E2 -19956.182} C_VEL
LIN {X 0,Y 267.901,Z 349.566,A -85,B 0,C 180,E1 -19958.907,E2 -19958.907} C_VEL
LIN {X 0,Y 267.085,Z 348.175,A -85,B 0,C 180,E1 -19959.709,E2 -19959.709} C_VEL
LIN {X 0,Y 264.382,Z 345.375,A -85,B 0,C 180,E1 -19962.581,E2 -19962.581} C_VEL
LIN {X 0,Y 263.08,Z 342.786,A -85,B 0,C 180,E1 -19964.507,E2 -19964.507} C_VEL
LIN {X 0,Y 259.999,Z 339.836,A -85,B 0,C 180,E1 -19972.233,E2 -19972.233} C_VEL
LIN {X 0,Y 259.942,Z 339.916,A -85,B 0,C 180,E1 -19974.81,E2 -19974.81} C_VEL
LIN {X 0,Y 260.882,Z 340.903,A -85,B 0,C 180,E1 -19978.843,E2 -19978.843} C_VEL
LIN {X 0,Y 263.439,Z 343.017,A -85,B 0,C 180,E1 -19983.432,E2 -19983.432} C_VEL
LIN {X 0,Y 265.222,Z 346.179,A -85,B 0,C 180,E1 -19985.835,E2 -19985.835} C_VEL
LIN {X 0,Y 267.453,Z 348.42,A -85,B 0,C 180,E1 -19988.063,E2 -19988.063} C_VEL
LIN {X 0,Y 269.65,Z 351.802,A -85,B 0,C 180,E1 -19990.039,E2 -19990.039} C_VEL
LIN {X 0,Y 271.283,Z 353.498,A -85,B 0,C 180,E1 -19991.282,E2 -19991.282} C_VEL
LIN {X 0,Y 274.164,Z 357.51,A -85,B 0,C 180,E1 -19993.34,E2 -19993.34} C_VEL
LIN {X 0,Y 278.411,Z 363.327,A -85,B 0,C 180,E1 -19995.953,E2 -19995.953} C_VEL
LIN {X 0,Y 281.975,Z 368.428,A -85,B 0,C 180,E1 -19997.904,E2 -19997.904} C_VEL
LIN {X 0,Y 286.565,Z 375.08,A -85,B 0,C 180,E1 -20000.164,E2 -20000.164} C_VEL
LIN {X 0,Y 293.161,Z 385.447,A -85,B 0,C 180,E1 -20003.045,E2 -20003.045} C_VEL
LIN {X 0,Y 299.383,Z 396.193,A -85,B 0,C 180,E1 -20005.484,E2 -20005.484} C_VEL
LIN {X 0,Y 297.384,Z 425.402,A -85,B 0,C 180,E1 -20006.167,E2 -20006.167} C_VEL
LIN {X 0,Y 292.125,Z 498.471,A -85,B 0,C 180,E1 -20007.854,E2 -20007.854} C_VEL
LIN {X 0,Y 289.877,Z 515.068,A -85,B 0,C 180,E1 -20008.402,E2 -20008.402} C_VEL
LIN {X 0,Y 287.06,Z 530.921,A -85,B 0,C 180,E1 -20009.195,E2 -20009.195} C_VEL
LIN {X 0,Y 283.568,Z 546.185,A -85,B 0,C 180,E1 -20010.191,E2 -20010.191} C_VEL
LIN {X 0,Y 279.233,Z 561.525,A -85,B 0,C 180,E1 -20011.459,E2 -20011.459} C_VEL
LIN {X 0,Y 274.347,Z 576.014,A -85,B 0,C 180,E1 -20012.969,E2 -20012.969} C_VEL
LIN {X 0,Y 269.241,Z 589.342,A -85,B 0,C 180,E1 -20014.691,E2 -20014.691} C_VEL
LIN {X 0,Y 263.864,Z 601.815,A -85,B 0,C 180,E1 -20016.642,E2 -20016.642} C_VEL
LIN {X 0,Y 258.505,Z 613.251,A -85,B 0,C 180,E1 -20018.83,E2 -20018.83} C_VEL
LIN {X 0,Y 252.866,Z 624.159,A -85,B 0,C 180,E1 -20021.373,E2 -20021.373} C_VEL
LIN {X 0,Y 247.425,Z 634.004,A -85,B 0,C 180,E1 -20024.174,E2 -20024.174} C_VEL
LIN {X 0,Y 242.654,Z 642.421,A -85,B 0,C 180,E1 -20027.107,E2 -20027.107} C_VEL
LIN {X 0,Y 237.837,Z 650.63,A -85,B 0,C 180,E1 -20030.694,E2 -20030.694} C_VEL
LIN {X 0,Y 234.024,Z 656.923,A -85,B 0,C 180,E1 -20034.18,E2 -20034.18} C_VEL
LIN {X 0,Y 230.954,Z 662.105,A -85,B 0,C 180,E1 -20037.824,E2 -20037.824} C_VEL
LIN {X 0,Y 228.128,Z 666.902,A -85,B 0,C 180,E1 -20042.476,E2 -20042.476} C_VEL
LIN {X 0,Y 226.695,Z 669.487,A -85,B 0,C 180,E1 -20046.232,E2 -20046.232} C_VEL
LIN {X 0,Y 225.813,Z 670.98,A -85,B 0,C 180,E1 -20049.979,E2 -20049.979} C_VEL
LIN {X 0,Y 225.411,Z 671.511,A -85,B 0,C 180,E1 -20053.703,E2 -20053.703} C_VEL
LIN {X 0,Y 225.356,Z 670.962,A -85,B 0,C 180,E1 -20057.39,E2 -20057.39} C_VEL
LIN {X 0,Y 225.435,Z 669.527,A -85,B 0,C 180,E1 -20061.032,E2 -20061.032} C_VEL
LIN {X 0,Y 225.975,Z 667.006,A -85,B 0,C 180,E1 -20064.646,E2 -20064.646} C_VEL
LIN {X 0,Y 226.513,Z 663.577,A -85,B 0,C 180,E1 -20068.222,E2 -20068.222} C_VEL
LIN {X 0,Y 227.63,Z 659.027,A -85,B 0,C 180,E1 -20071.769,E2 -20071.769} C_VEL
LIN {X 0,Y 229.239,Z 653.391,A -85,B 0,C 180,E1 -20075.277,E2 -20075.277} C_VEL
LIN {X 0,Y 231.536,Z 646.557,A -85,B 0,C 180,E1 -20078.729,E2 -20078.729} C_VEL
LIN {X 0,Y 234.538,Z 638.255,A -85,B 0,C 180,E1 -20082.108,E2 -20082.108} C_VEL
LIN {X 0,Y 238.193,Z 628.401,A -85,B 0,C 180,E1 -20085.399,E2 -20085.399} C_VEL
LIN {X 0,Y 241.915,Z 618.279,A -85,B 0,C 180,E1 -20088.198,E2 -20088.198} C_VEL
LIN {X 0,Y 245.956,Z 606.45,A -85,B 0,C 180,E1 -20090.927,E2 -20090.927} C_VEL
LIN {X 0,Y 250.136,Z 593.419,A -85,B 0,C 180,E1 -20093.382,E2 -20093.382} C_VEL
LIN {X 0,Y 253.977,Z 580.408,A -85,B 0,C 180,E1 -20095.398,E2 -20095.398} C_VEL
LIN {X 0,Y 257.772,Z 566.433,A -85,B 0,C 180,E1 -20097.173,E2 -20097.173} C_VEL
LIN {X 0,Y 261.214,Z 551.353,A -85,B 0,C 180,E1 -20098.746,E2 -20098.746} C_VEL
LIN {X 0,Y 263.833,Z 537.96,A -85,B 0,C 180,E1 -20099.854,E2 -20099.854} C_VEL
LIN {X 0,Y 266.498,Z 521.755,A -85,B 0,C 180,E1 -20100.892,E2 -20100.892} C_VEL
LIN {X 0,Y 268.628,Z 504.955,A -85,B 0,C 180,E1 -20101.66,E2 -20101.66} C_VEL
LIN {X 0,Y 270.018,Z 487.499,A -85,B 0,C 180,E1 -20102.192,E2 -20102.192} C_VEL
LIN {X 0,Y 276.032,Z 380.613,A -85,B 0,C 180,E1 -20104.797,E2 -20104.797} C_VEL
LIN {X 0,Y 274.398,Z 376.982,A -85,B 0,C 180,E1 -20105.246,E2 -20105.246} C_VEL
LIN {X 0,Y 266.147,Z 361.85,A -85,B 0,C 180,E1 -20107.522,E2 -20107.522} C_VEL
LIN {X 0,Y 258.332,Z 348.837,A -85,B 0,C 180,E1 -20109.849,E2 -20109.849} C_VEL
LIN {X 0,Y 251.196,Z 337.996,A -85,B 0,C 180,E1 -20112.148,E2 -20112.148} C_VEL
LIN {X 0,Y 245.333,Z 329.901,A -85,B 0,C 180,E1 -20114.186,E2 -20114.186} C_VEL
LIN {X 0,Y 242.261,Z 325.779,A -85,B 0,C 180,E1 -20115.327,E2 -20115.327} C_VEL
LIN {X 0,Y 239.104,Z 321.549,A -85,B 0,C 180,E1 -20116.56,E2 -20116.56} C_VEL
LIN {X 0,Y 236.457,Z 318.218,A -85,B 0,C 180,E1 -20117.633,E2 -20117.633} C_VEL
LIN {X 0,Y 235.565,Z 316.953,A -85,B 0,C 180,E1 -20118.015,E2 -20118.015} C_VEL
LIN {X 0,Y 233.005,Z 314.171,A -85,B 0,C 180,E1 -20119.1,E2 -20119.1} C_VEL
LIN {X 0,Y 231.706,Z 311.852,A -85,B 0,C 180,E1 -20119.724,E2 -20119.724} C_VEL
LIN {X 0,Y 229.407,Z 309.976,A -85,B 0,C 180,E1 -20120.741,E2 -20120.741} C_VEL
LIN {X 0,Y 228.044,Z 307.343,A -85,B 0,C 180,E1 -20121.461,E2 -20121.461} C_VEL
LIN {X 0,Y 227.844,Z 306.355,A -85,B 0,C 180,E1 -20121.664,E2 -20121.664} C_VEL
LIN {X 0,Y 227.878,Z 306.376,A -85,B 0,C 180,E1 -20126.378,E2 -20126.378} C_VEL
LIN {X 0,Y 227.874,Z 306.391,A -85,B 0,C 180,E1 -20130.43,E2 -20130.43} C_VEL
LIN {X 0,Y 227.903,Z 306.401,A -85,B 0,C 180,E1 -20134.422,E2 -20134.422} C_VEL
LIN {X 0,Y 227.953,Z 306.396,A -85,B 0,C 180,E1 -20138.285,E2 -20138.285} C_VEL
LIN {X 0,Y 228.025,Z 306.383,A -85,B 0,C 180,E1 -20143.894,E2 -20143.894} C_VEL
LIN {X 0,Y 228.068,Z 306.365,A -85,B 0,C 180,E1 -20147.542,E2 -20147.542} C_VEL
LIN {X 0,Y 228.258,Z 306.362,A -85,B 0,C 180,E1 -20151.371,E2 -20151.371} C_VEL
LIN {X 0,Y 227.599,Z 306.431,A -85,B 0,C 180,E1 -20152.843,E2 -20152.843} C_VEL
LIN {X 0,Y 224.835,Z 306.774,A -85,B 0,C 180,E1 -20155.248,E2 -20155.248} C_VEL
LIN {X 0,Y 222.524,Z 307.08,A -85,B 0,C 180,E1 -20157.21,E2 -20157.21} C_VEL
LIN {X 0,Y 221.577,Z 307.183,A -85,B 0,C 180,E1 -20158.73,E2 -20158.73} C_VEL
LIN {X 0,Y 221.523,Z 307.183,A -85,B 0,C 180,E1 -20159.244,E2 -20159.244} C_VEL
LIN {X 0,Y 221.512,Z 307.187,A -85,B 0,C 180,E1 -20161.817,E2 -20161.817} C_VEL
LIN {X 0,Y 221.257,Z 307.198,A -85,B 0,C 180,E1 -20167.299,E2 -20167.299} C_VEL
LIN {X 0,Y 221.066,Z 307.261,A -85,B 0,C 180,E1 -20170.995,E2 -20170.995} C_VEL
LIN {X 0,Y 221.006,Z 307.265,A -85,B 0,C 180,E1 -20176.63,E2 -20176.63} C_VEL
LIN {X 0,Y 220.935,Z 307.345,A -85,B 0,C 180,E1 -20181.947,E2 -20181.947} C_VEL
LIN {X 0,Y 221.63,Z 309.69,A -85,B 0,C 180,E1 -20182.444,E2 -20182.444} C_VEL
LIN {X 0,Y 223.385,Z 311.87,A -85,B 0,C 180,E1 -20183.409,E2 -20183.409} C_VEL
LIN {X 0,Y 225.306,Z 313.196,A -85,B 0,C 180,E1 -20184.351,E2 -20184.351} C_VEL
LIN {X 0,Y 227.102,Z 316.267,A -85,B 0,C 180,E1 -20185.305,E2 -20185.305} C_VEL
LIN {X 0,Y 229.555,Z 318.636,A -85,B 0,C 180,E1 -20186.438,E2 -20186.438} C_VEL
LIN {X 0,Y 231.959,Z 322.089,A -85,B 0,C 180,E1 -20187.557,E2 -20187.557} C_VEL
LIN {X 0,Y 233.529,Z 323.765,A -85,B 0,C 180,E1 -20188.232,E2 -20188.232} C_VEL
LIN {X 0,Y 236.608,Z 327.798,A -85,B 0,C 180,E1 -20189.536,E2 -20189.536} C_VEL
LIN {X 0,Y 243.919,Z 337.826,A -85,B 0,C 180,E1 -20192.378,E2 -20192.378} C_VEL
LIN {X 0,Y 248.746,Z 345.002,A -85,B 0,C 180,E1 -20194.1,E2 -20194.1} C_VEL
LIN {X 0,Y 255.532,Z 357.16,A -85,B 0,C 180,E1 -20196.418,E2 -20196.418} C_VEL
LIN {X 0,Y 262.229,Z 370.328,A -85,B 0,C 180,E1 -20198.544,E2 -20198.544} C_VEL
LIN {X 0,Y 268.158,Z 383.389,A -85,B 0,C 180,E1 -20200.332,E2 -20200.332} C_VEL
LIN {X 0,Y 270.528,Z 388.896,A -85,B 0,C 180,E1 -20201.022,E2 -20201.022} C_VEL
LIN {X 0,Y 263.461,Z 510.105,A -85,B 0,C 180,E1 -20204.064,E2 -20204.064} C_VEL
LIN {X 0,Y 261.544,Z 526.913,A -85,B 0,C 180,E1 -20204.732,E2 -20204.732} C_VEL
LIN {X 0,Y 258.868,Z 543.314,A -85,B 0,C 180,E1 -20205.646,E2 -20205.646} C_VEL
LIN {X 0,Y 255.64,Z 559.352,A -85,B 0,C 180,E1 -20206.854,E2 -20206.854} C_VEL
LIN {X 0,Y 252.063,Z 574.115,A -85,B 0,C 180,E1 -20208.266,E2 -20208.266} C_VEL
LIN {X 0,Y 248.193,Z 587.998,A -85,B 0,C 180,E1 -20209.917,E2 -20209.917} C_VEL
LIN {X 0,Y 243.929,Z 601.975,A -85,B 0,C 180,E1 -20211.987,E2 -20211.987} C_VEL
LIN {X 0,Y 239.968,Z 613.99,A -85,B 0,C 180,E1 -20214.145,E2 -20214.145} C_VEL
LIN {X 0,Y 235.591,Z 626.194,A -85,B 0,C 180,E1 -20216.769,E2 -20216.769} C_VEL
LIN {X 0,Y 231.255,Z 638.047,A -85,B 0,C 180,E1 -20219.904,E2 -20219.904} C_VEL
LIN {X 0,Y 227.338,Z 648.658,A -85,B 0,C 180,E1 -20223.369,E2 -20223.369} C_VEL
LIN {X 0,Y 224.245,Z 657.509,A -85,B 0,C 180,E1 -20226.936,E2 -20226.936} C_VEL
LIN {X 0,Y 221.788,Z 664.876,A -85,B 0,C 180,E1 -20230.566,E2 -20230.566} C_VEL
LIN {X 0,Y 220.165,Z 670.97,A -85,B 0,C 180,E1 -20234.257,E2 -20234.257} C_VEL
LIN {X 0,Y 218.914,Z 676.832,A -85,B 0,C 180,E1 -20238.894,E2 -20238.894} C_VEL
LIN {X 0,Y 218.575,Z 680.223,A -85,B 0,C 180,E1 -20242.611,E2 -20242.611} C_VEL
LIN {X 0,Y 218.518,Z 682.628,A -85,B 0,C 180,E1 -20246.312,E2 -20246.312} C_VEL
LIN {X 0,Y 218.646,Z 683.957,A -85,B 0,C 180,E1 -20250,E2 -20250} C_VEL
LIN {X 0,Y 218.475,Z 684.349,A -85,B 0,C 180,E1 -20253.689,E2 -20253.689} C_VEL
LIN {X 0,Y 218.526,Z 683.715,A -85,B 0,C 180,E1 -20257.391,E2 -20257.391} C_VEL
LIN {X 0,Y 218.969,Z 682.202,A -85,B 0,C 180,E1 -20261.103,E2 -20261.103} C_VEL
LIN {X 0,Y 220.05,Z 679.652,A -85,B 0,C 180,E1 -20264.804,E2 -20264.804} C_VEL
LIN {X 0,Y 222.33,Z 675.115,A -85,B 0,C 180,E1 -20269.385,E2 -20269.385} C_VEL
LIN {X 0,Y 225.029,Z 670.357,A -85,B 0,C 180,E1 -20272.979,E2 -20272.979} C_VEL
LIN {X 0,Y 229.459,Z 662.758,A -85,B 0,C 180,E1 -20277.35,E2 -20277.35} C_VEL
LIN {X 0,Y 234.595,Z 654.22,A -85,B 0,C 180,E1 -20281.117,E2 -20281.117} C_VEL
LIN {X 0,Y 239.269,Z 646.299,A -85,B 0,C 180,E1 -20283.924,E2 -20283.924} C_VEL
LIN {X 0,Y 244.409,Z 637.199,A -85,B 0,C 180,E1 -20286.633,E2 -20286.633} C_VEL
LIN {X 0,Y 250.103,Z 626.501,A -85,B 0,C 180,E1 -20289.217,E2 -20289.217} C_VEL
LIN {X 0,Y 256.457,Z 613.978,A -85,B 0,C 180,E1 -20291.648,E2 -20291.648} C_VEL
LIN {X 0,Y 262.41,Z 600.763,A -85,B 0,C 180,E1 -20293.751,E2 -20293.751} C_VEL
LIN {X 0,Y 267.771,Z 587.898,A -85,B 0,C 180,E1 -20295.392,E2 -20295.392} C_VEL
LIN {X 0,Y 273.077,Z 573.147,A -85,B 0,C 180,E1 -20296.909,E2 -20296.909} C_VEL
LIN {X 0,Y 277.997,Z 556.942,A -85,B 0,C 180,E1 -20298.227,E2 -20298.227} C_VEL
LIN {X 0,Y 282.012,Z 541.046,A -85,B 0,C 180,E1 -20299.198,E2 -20299.198} C_VEL
LIN {X 0,Y 285.29,Z 524.186,A -85,B 0,C 180,E1 -20299.969,E2 -20299.969} C_VEL
LIN {X 0,Y 287.619,Z 507.196,A -85,B 0,C 180,E1 -20300.501,E2 -20300.501} C_VEL
LIN {X 0,Y 295.095,Z 404.799,A -85,B 0,C 180,E1 -20302.874,E2 -20302.874} C_VEL
LIN {X 0,Y 289.938,Z 394.123,A -85,B 0,C 180,E1 -20305.071,E2 -20305.071} C_VEL
LIN {X 0,Y 285.118,Z 385.088,A -85,B 0,C 180,E1 -20307.299,E2 -20307.299} C_VEL
LIN {X 0,Y 280.599,Z 377.017,A -85,B 0,C 180,E1 -20309.628,E2 -20309.628} C_VEL
LIN {X 0,Y 275.953,Z 369.431,A -85,B 0,C 180,E1 -20312.304,E2 -20312.304} C_VEL
LIN {X 0,Y 272.516,Z 364.112,A -85,B 0,C 180,E1 -20314.551,E2 -20314.551} C_VEL
LIN {X 0,Y 269.135,Z 359.576,A -85,B 0,C 180,E1 -20317.064,E2 -20317.064} C_VEL
LIN {X 0,Y 266.405,Z 356.051,A -85,B 0,C 180,E1 -20319.437,E2 -20319.437} C_VEL
LIN {X 0,Y 265.728,Z 354.951,A -85,B 0,C 180,E1 -20320.122,E2 -20320.122} C_VEL
LIN {X 0,Y 263.205,Z 352.202,A -85,B 0,C 180,E1 -20322.92,E2 -20322.92} C_VEL
LIN {X 0,Y 261.958,Z 349.713,A -85,B 0,C 180,E1 -20324.837,E2 -20324.837} C_VEL
LIN {X 0,Y 259.124,Z 346.902,A -85,B 0,C 180,E1 -20332.207,E2 -20332.207} C_VEL
LIN {X 0,Y 259.067,Z 346.94,A -85,B 0,C 180,E1 -20334.793,E2 -20334.793} C_VEL
LIN {X 0,Y 260.074,Z 348.046,A -85,B 0,C 180,E1 -20339.04,E2 -20339.04} C_VEL
LIN {X 0,Y 262.381,Z 350.055,A -85,B 0,C 180,E1 -20343.221,E2 -20343.221} C_VEL
LIN {X 0,Y 264.213,Z 353.276,A -85,B 0,C 180,E1 -20345.732,E2 -20345.732} C_VEL
LIN {X 0,Y 266.099,Z 355.181,A -85,B 0,C 180,E1 -20347.663,E2 -20347.663} C_VEL
LIN {X 0,Y 268.329,Z 358.63,A -85,B 0,C 180,E1 -20349.732,E2 -20349.732} C_VEL
LIN {X 0,Y 269.851,Z 360.352,A -85,B 0,C 180,E1 -20350.932,E2 -20350.932} C_VEL
LIN {X 0,Y 273.771,Z 365.874,A -85,B 0,C 180,E1 -20353.737,E2 -20353.737} C_VEL
LIN {X 0,Y 276.852,Z 370.262,A -85,B 0,C 180,E1 -20355.647,E2 -20355.647} C_VEL
LIN {X 0,Y 279.888,Z 374.675,A -85,B 0,C 180,E1 -20357.359,E2 -20357.359} C_VEL
LIN {X 0,Y 284.449,Z 381.449,A -85,B 0,C 180,E1 -20359.683,E2 -20359.683} C_VEL
LIN {X 0,Y 290.669,Z 391.501,A -85,B 0,C 180,E1 -20362.496,E2 -20362.496} C_VEL
LIN {X 0,Y 295.405,Z 399.766,A -85,B 0,C 180,E1 -20364.439,E2 -20364.439} C_VEL
LIN {X 0,Y 287.957,Z 499.687,A -85,B 0,C 180,E1 -20366.731,E2 -20366.731} C_VEL
LIN {X 0,Y 285.523,Z 516.885,A -85,B 0,C 180,E1 -20367.323,E2 -20367.323} C_VEL
LIN {X 0,Y 282.425,Z 533.225,A -85,B 0,C 180,E1 -20368.171,E2 -20368.171} C_VEL
LIN {X 0,Y 278.735,Z 548.296,A -85,B 0,C 180,E1 -20369.187,E2 -20369.187} C_VEL
LIN {X 0,Y 274.757,Z 561.806,A -85,B 0,C 180,E1 -20370.312,E2 -20370.312} C_VEL
LIN {X 0,Y 269.795,Z 576.071,A -85,B 0,C 180,E1 -20371.803,E2 -20371.803} C_VEL
LIN {X 0,Y 264.517,Z 589.409,A -85,B 0,C 180,E1 -20373.528,E2 -20373.528} C_VEL
LIN {X 0,Y 258.948,Z 601.905,A -85,B 0,C 180,E1 -20375.49,E2 -20375.49} C_VEL
LIN {X 0,Y 253.212,Z 613.684,A -85,B 0,C 180,E1 -20377.761,E2 -20377.761} C_VEL
LIN {X 0,Y 247.25,Z 624.741,A -85,B 0,C 180,E1 -20380.379,E2 -20380.379} C_VEL
LIN {X 0,Y 241.435,Z 634.777,A -85,B 0,C 180,E1 -20383.303,E2 -20383.303} C_VEL
LIN {X 0,Y 235.795,Z 644.135,A -85,B 0,C 180,E1 -20386.722,E2 -20386.722} C_VEL
LIN {X 0,Y 230.998,Z 651.873,A -85,B 0,C 180,E1 -20390.289,E2 -20390.289} C_VEL
LIN {X 0,Y 227.007,Z 658.146,A -85,B 0,C 180,E1 -20393.968,E2 -20393.968} C_VEL
LIN {X 0,Y 223.623,Z 663.457,A -85,B 0,C 180,E1 -20398.057,E2 -20398.057} C_VEL
LIN {X 0,Y 221.455,Z 666.902,A -85,B 0,C 180,E1 -20401.573,E2 -20401.573} C_VEL
LIN {X 0,Y 219.827,Z 669.537,A -85,B 0,C 180,E1 -20405.442,E2 -20405.442} C_VEL
LIN {X 0,Y 218.839,Z 671.125,A -85,B 0,C 180,E1 -20409.313,E2 -20409.313} C_VEL
LIN {X 0,Y 218.355,Z 671.701,A -85,B 0,C 180,E1 -20413.161,E2 -20413.161} C_VEL
LIN {X 0,Y 218.246,Z 671.244,A -85,B 0,C 180,E1 -20416.972,E2 -20416.972} C_VEL
LIN {X 0,Y 218.327,Z 669.862,A -85,B 0,C 180,E1 -20420.738,E2 -20420.738} C_VEL
LIN {X 0,Y 218.866,Z 667.371,A -85,B 0,C 180,E1 -20424.538,E2 -20424.538} C_VEL
LIN {X 0,Y 219.4,Z 664.08,A -85,B 0,C 180,E1 -20428.164,E2 -20428.164} C_VEL
LIN {X 0,Y 220.559,Z 659.585,A -85,B 0,C 180,E1 -20431.826,E2 -20431.826} C_VEL
LIN {X 0,Y 222.181,Z 654.054,A -85,B 0,C 180,E1 -20435.445,E2 -20435.445} C_VEL
LIN {X 0,Y 224.543,Z 647.272,A -85,B 0,C 180,E1 -20439.003,E2 -20439.003} C_VEL
LIN {X 0,Y 227.63,Z 639.089,A -85,B 0,C 180,E1 -20442.481,E2 -20442.481} C_VEL
LIN {X 0,Y 231.411,Z 629.364,A -85,B 0,C 180,E1 -20445.862,E2 -20445.862} C_VEL
LIN {X 0,Y 235.219,Z 619.399,A -85,B 0,C 180,E1 -20448.735,E2 -20448.735} C_VEL
LIN {X 0,Y 239.417,Z 607.659,A -85,B 0,C 180,E1 -20451.526,E2 -20451.526} C_VEL
LIN {X 0,Y 243.357,Z 595.873,A -85,B 0,C 180,E1 -20453.848,E2 -20453.848} C_VEL
LIN {X 0,Y 247.258,Z 583.336,A -85,B 0,C 180,E1 -20455.913,E2 -20455.913} C_VEL
LIN {X 0,Y 251.145,Z 569.895,A -85,B 0,C 180,E1 -20457.725,E2 -20457.725} C_VEL
LIN {X 0,Y 254.684,Z 555.382,A -85,B 0,C 180,E1 -20459.328,E2 -20459.328} C_VEL
LIN {X 0,Y 257.771,Z 540.682,A -85,B 0,C 180,E1 -20460.631,E2 -20460.631} C_VEL
LIN {X 0,Y 260.684,Z 524.553,A -85,B 0,C 180,E1 -20461.716,E2 -20461.716} C_VEL
LIN {X 0,Y 262.809,Z 508.904,A -85,B 0,C 180,E1 -20462.503,E2 -20462.503} C_VEL
LIN {X 0,Y 264.301,Z 493.119,A -85,B 0,C 180,E1 -20463.032,E2 -20463.032} C_VEL
LIN {X 0,Y 270.735,Z 382.823,A -85,B 0,C 180,E1 -20465.77,E2 -20465.77} C_VEL
LIN {X 0,Y 262.934,Z 368.07,A -85,B 0,C 180,E1 -20467.998,E2 -20467.998} C_VEL
LIN {X 0,Y 254.894,Z 354.38,A -85,B 0,C 180,E1 -20470.475,E2 -20470.475} C_VEL
LIN {X 0,Y 247.894,Z 343.605,A -85,B 0,C 180,E1 -20472.811,E2 -20472.811} C_VEL
LIN {X 0,Y 241.811,Z 335.072,A -85,B 0,C 180,E1 -20475.015,E2 -20475.015} C_VEL
LIN {X 0,Y 238.902,Z 331.097,A -85,B 0,C 180,E1 -20476.143,E2 -20476.143} C_VEL
LIN {X 0,Y 235.996,Z 327.244,A -85,B 0,C 180,E1 -20477.319,E2 -20477.319} C_VEL
LIN {X 0,Y 232.542,Z 322.732,A -85,B 0,C 180,E1 -20478.798,E2 -20478.798} C_VEL
LIN {X 0,Y 229.916,Z 319.478,A -85,B 0,C 180,E1 -20479.983,E2 -20479.983} C_VEL
LIN {X 0,Y 228.925,Z 318.024,A -85,B 0,C 180,E1 -20480.462,E2 -20480.462} C_VEL
LIN {X 0,Y 226.359,Z 315.323,A -85,B 0,C 180,E1 -20481.683,E2 -20481.683} C_VEL
LIN {X 0,Y 224.925,Z 312.803,A -85,B 0,C 180,E1 -20482.46,E2 -20482.46} C_VEL
LIN {X 0,Y 222.391,Z 310.865,A -85,B 0,C 180,E1 -20483.732,E2 -20483.732} C_VEL
LIN {X 0,Y 221.054,Z 308.416,A -85,B 0,C 180,E1 -20484.532,E2 -20484.532} C_VEL
LIN {X 0,Y 220.786,Z 307.227,A -85,B 0,C 180,E1 -20484.762,E2 -20484.762} C_VEL
LIN {X 0,Y 220.836,Z 307.276,A -85,B 0,C 180,E1 -20489.389,E2 -20489.389} C_VEL
LIN {X 0,Y 220.876,Z 307.286,A -85,B 0,C 180,E1 -20493.546,E2 -20493.546} C_VEL
LIN {X 0,Y 220.867,Z 307.268,A -85,B 0,C 180,E1 -20497.551,E2 -20497.551} C_VEL
LIN {X 0,Y 220.931,Z 307.253,A -85,B 0,C 180,E1 -20502.616,E2 -20502.616} C_VEL
LIN {X 0,Y 221.005,Z 307.247,A -85,B 0,C 180,E1 -20507.137,E2 -20507.137} C_VEL
LIN {X 0,Y 221.193,Z 307.237,A -85,B 0,C 180,E1 -20511.372,E2 -20511.372} C_VEL
LIN {X 0,Y 221.126,Z 307.227,A -85,B 0,C 180,E1 -20514.528,E2 -20514.528} C_VEL
LIN {X 0,Y 221.507,Z 307.2,A -85,B 0,C 180,E1 -20518.181,E2 -20518.181} C_VEL
LIN {X 0,Y 221.523,Z 307.183,A -85,B 0,C 180,E1 -20519.244,E2 -20519.244} C_VEL
LIN {X 0,Y 220.856,Z 307.267,A -85,B 0,C 180,E1 -20520.758,E2 -20520.758} C_VEL
LIN {X 0,Y 219.176,Z 307.492,A -85,B 0,C 180,E1 -20522.241,E2 -20522.241} C_VEL
LIN {X 0,Y 215.24,Z 307.965,A -85,B 0,C 180,E1 -20525.232,E2 -20525.232} C_VEL
LIN {X 0,Y 214.214,Z 308.076,A -85,B 0,C 180,E1 -20526.803,E2 -20526.803} C_VEL
LIN {X 0,Y 214.175,Z 308.08,A -85,B 0,C 180,E1 -20527.336,E2 -20527.336} C_VEL
LIN {X 0,Y 213.997,Z 308.138,A -85,B 0,C 180,E1 -20531.363,E2 -20531.363} C_VEL
LIN {X 0,Y 213.92,Z 308.146,A -85,B 0,C 180,E1 -20535.237,E2 -20535.237} C_VEL
LIN {X 0,Y 213.888,Z 308.181,A -85,B 0,C 180,E1 -20538.218,E2 -20538.218} C_VEL
LIN {X 0,Y 214.596,Z 310.505,A -85,B 0,C 180,E1 -20538.815,E2 -20538.815} C_VEL
LIN {X 0,Y 216.316,Z 312.728,A -85,B 0,C 180,E1 -20539.945,E2 -20539.945} C_VEL
LIN {X 0,Y 218.515,Z 314.142,A -85,B 0,C 180,E1 -20541.212,E2 -20541.212} C_VEL
LIN {X 0,Y 220.164,Z 317.147,A -85,B 0,C 180,E1 -20542.245,E2 -20542.245} C_VEL
LIN {X 0,Y 223.023,Z 319.852,A -85,B 0,C 180,E1 -20543.762,E2 -20543.762} C_VEL
LIN {X 0,Y 225.328,Z 323.139,A -85,B 0,C 180,E1 -20544.978,E2 -20544.978} C_VEL
LIN {X 0,Y 227.136,Z 325.074,A -85,B 0,C 180,E1 -20545.847,E2 -20545.847} C_VEL
LIN {X 0,Y 229.913,Z 328.708,A -85,B 0,C 180,E1 -20547.155,E2 -20547.155} C_VEL
LIN {X 0,Y 234.773,Z 335.212,A -85,B 0,C 180,E1 -20549.291,E2 -20549.291} C_VEL
LIN {X 0,Y 240.442,Z 342.97,A -85,B 0,C 180,E1 -20551.559,E2 -20551.559} C_VEL
LIN {X 0,Y 245.345,Z 350.469,A -85,B 0,C 180,E1 -20553.387,E2 -20553.387} C_VEL
LIN {X 0,Y 251.561,Z 361.783,A -85,B 0,C 180,E1 -20555.598,E2 -20555.598} C_VEL
LIN {X 0,Y 257.875,Z 374.424,A -85,B 0,C 180,E1 -20557.697,E2 -20557.697} C_VEL
LIN {X 0,Y 263.841,Z 387.781,A -85,B 0,C 180,E1 -20559.576,E2 -20559.576} C_VEL
LIN {X 0,Y 265.299,Z 391.235,A -85,B 0,C 180,E1 -20560.021,E2 -20560.021} C_VEL
LIN {X 0,Y 258.163,Z 509.46,A -85,B 0,C 180,E1 -20563.02,E2 -20563.02} C_VEL
LIN {X 0,Y 256.218,Z 526.378,A -85,B 0,C 180,E1 -20563.695,E2 -20563.695} C_VEL
LIN {X 0,Y 253.525,Z 542.544,A -85,B 0,C 180,E1 -20564.595,E2 -20564.595} C_VEL
LIN {X 0,Y 250.421,Z 557.708,A -85,B 0,C 180,E1 -20565.725,E2 -20565.725} C_VEL
LIN {X 0,Y 246.743,Z 572.772,A -85,B 0,C 180,E1 -20567.154,E2 -20567.154} C_VEL
LIN {X 0,Y 243.103,Z 585.474,A -85,B 0,C 180,E1 -20568.654,E2 -20568.654} C_VEL
LIN {X 0,Y 238.701,Z 599.74,A -85,B 0,C 180,E1 -20570.727,E2 -20570.727} C_VEL
LIN {X 0,Y 234.456,Z 612.088,A -85,B 0,C 180,E1 -20572.896,E2 -20572.896} C_VEL
LIN {X 0,Y 229.678,Z 625.113,A -85,B 0,C 180,E1 -20575.707,E2 -20575.707} C_VEL
LIN {X 0,Y 225.044,Z 637.331,A -85,B 0,C 180,E1 -20578.984,E2 -20578.984} C_VEL
LIN {X 0,Y 221.33,Z 646.747,A -85,B 0,C 180,E1 -20582.072,E2 -20582.072} C_VEL
LIN {X 0,Y 217.955,Z 655.91,A -85,B 0,C 180,E1 -20585.725,E2 -20585.725} C_VEL
LIN {X 0,Y 215.561,Z 662.687,A -85,B 0,C 180,E1 -20588.984,E2 -20588.984} C_VEL
LIN {X 0,Y 213.567,Z 669.071,A -85,B 0,C 180,E1 -20592.773,E2 -20592.773} C_VEL
LIN {X 0,Y 212.328,Z 674.276,A -85,B 0,C 180,E1 -20596.603,E2 -20596.603} C_VEL
LIN {X 0,Y 211.603,Z 678.295,A -85,B 0,C 180,E1 -20600.441,E2 -20600.441} C_VEL
LIN {X 0,Y 211.471,Z 681.24,A -85,B 0,C 180,E1 -20604.278,E2 -20604.278} C_VEL
LIN {X 0,Y 211.463,Z 683.152,A -85,B 0,C 180,E1 -20608.096,E2 -20608.096} C_VEL
LIN {X 0,Y 211.561,Z 683.709,A -85,B 0,C 180,E1 -20610,E2 -20610} C_VEL
LIN {X 0,Y 211.39,Z 684.122,A -85,B 0,C 180,E1 -20614.145,E2 -20614.145} C_VEL
LIN {X 0,Y 211.438,Z 683.547,A -85,B 0,C 180,E1 -20617.641,E2 -20617.641} C_VEL
LIN {X 0,Y 211.929,Z 682.082,A -85,B 0,C 180,E1 -20621.477,E2 -20621.477} C_VEL
LIN {X 0,Y 213.099,Z 679.566,A -85,B 0,C 180,E1 -20625.298,E2 -20625.298} C_VEL
LIN {X 0,Y 215.545,Z 675.088,A -85,B 0,C 180,E1 -20630.021,E2 -20630.021} C_VEL
LIN {X 0,Y 218.418,Z 670.374,A -85,B 0,C 180,E1 -20633.717,E2 -20633.717} C_VEL
LIN {X 0,Y 223.097,Z 662.845,A -85,B 0,C 180,E1 -20638.199,E2 -20638.199} C_VEL
LIN {X 0,Y 228.482,Z 654.371,A -85,B 0,C 180,E1 -20642.046,E2 -20642.046} C_VEL
LIN {X 0,Y 234.127,Z 645.304,A -85,B 0,C 180,E1 -20645.299,E2 -20645.299} C_VEL
LIN {X 0,Y 239.536,Z 636.055,A -85,B 0,C 180,E1 -20648.035,E2 -20648.035} C_VEL
LIN {X 0,Y 245.522,Z 625.263,A -85,B 0,C 180,E1 -20650.633,E2 -20650.633} C_VEL
LIN {X 0,Y 252.193,Z 612.546,A -85,B 0,C 180,E1 -20653.06,E2 -20653.06} C_VEL
LIN {X 0,Y 257.323,Z 601.48,A -85,B 0,C 180,E1 -20654.83,E2 -20654.83} C_VEL
LIN {X 0,Y 263.436,Z 587.323,A -85,B 0,C 180,E1 -20656.634,E2 -20656.634} C_VEL
LIN {X 0,Y 268.892,Z 572.531,A -85,B 0,C 180,E1 -20658.151,E2 -20658.151} C_VEL
LIN {X 0,Y 273.381,Z 558.177,A -85,B 0,C 180,E1 -20659.322,E2 -20659.322} C_VEL
LIN {X 0,Y 277.469,Z 542.732,A -85,B 0,C 180,E1 -20660.298,E2 -20660.298} C_VEL
LIN {X 0,Y 280.879,Z 526.404,A -85,B 0,C 180,E1 -20661.07,E2 -20661.07} C_VEL
LIN {X 0,Y 283.324,Z 510.125,A -85,B 0,C 180,E1 -20661.614,E2 -20661.614} C_VEL
LIN {X 0,Y 286.751,Z 466.785,A -85,B 0,C 180,E1 -20662.639,E2 -20662.639} C_VEL
LIN {X 0,Y 291.105,Z 407.946,A -85,B 0,C 180,E1 -20664.006,E2 -20664.006} C_VEL
LIN {X 0,Y 286.222,Z 397.713,A -85,B 0,C 180,E1 -20666.214,E2 -20666.214} C_VEL
LIN {X 0,Y 281.694,Z 389.141,A -85,B 0,C 180,E1 -20668.449,E2 -20668.449} C_VEL
LIN {X 0,Y 277.93,Z 382.247,A -85,B 0,C 180,E1 -20670.509,E2 -20670.509} C_VEL
LIN {X 0,Y 273.616,Z 375.119,A -85,B 0,C 180,E1 -20673.125,E2 -20673.125} C_VEL
LIN {X 0,Y 270.786,Z 370.584,A -85,B 0,C 180,E1 -20675.073,E2 -20675.073} C_VEL
LIN {X 0,Y 267.55,Z 366.135,A -85,B 0,C 180,E1 -20677.575,E2 -20677.575} C_VEL
LIN {X 0,Y 264.907,Z 362.483,A -85,B 0,C 180,E1 -20680,E2 -20680} C_VEL
LIN {X 0,Y 263.856,Z 361.286,A -85,B 0,C 180,E1 -20681.073,E2 -20681.073} C_VEL
LIN {X 0,Y 261.536,Z 358.063,A -85,B 0,C 180,E1 -20684.013,E2 -20684.013} C_VEL
LIN {X 0,Y 260.875,Z 356.694,A -85,B 0,C 180,E1 -20685.118,E2 -20685.118} C_VEL
LIN {X 0,Y 258.249,Z 353.966,A -85,B 0,C 180,E1 -20692.18,E2 -20692.18} C_VEL
LIN {X 0,Y 258.189,Z 353.989,A -85,B 0,C 180,E1 -20694.775,E2 -20694.775} C_VEL
LIN {X 0,Y 259.215,Z 355.137,A -85,B 0,C 180,E1 -20699.104,E2 -20699.104} C_VEL
LIN {X 0,Y 261.313,Z 357.083,A -85,B 0,C 180,E1 -20702.988,E2 -20702.988} C_VEL
LIN {X 0,Y 263.535,Z 360.716,A -85,B 0,C 180,E1 -20705.998,E2 -20705.998} C_VEL
LIN {X 0,Y 264.821,Z 362.074,A -85,B 0,C 180,E1 -20707.327,E2 -20707.327} C_VEL
LIN {X 0,Y 267.126,Z 365.579,A -85,B 0,C 180,E1 -20709.513,E2 -20709.513} C_VEL
LIN {X 0,Y 268.346,Z 367.019,A -85,B 0,C 180,E1 -20710.505,E2 -20710.505} C_VEL
LIN {X 0,Y 272.069,Z 372.398,A -85,B 0,C 180,E1 -20713.27,E2 -20713.27} C_VEL
LIN {X 0,Y 275.15,Z 376.923,A -85,B 0,C 180,E1 -20715.244,E2 -20715.244} C_VEL
LIN {X 0,Y 279.726,Z 383.674,A -85,B 0,C 180,E1 -20717.834,E2 -20717.834} C_VEL
LIN {X 0,Y 285.81,Z 393.459,A -85,B 0,C 180,E1 -20720.856,E2 -20720.856} C_VEL
LIN {X 0,Y 291.421,Z 403.311,A -85,B 0,C 180,E1 -20723.323,E2 -20723.323} C_VEL
LIN {X 0,Y 284.068,Z 499.393,A -85,B 0,C 180,E1 -20725.543,E2 -20725.543} C_VEL
LIN {X 0,Y 281.698,Z 515.784,A -85,B 0,C 180,E1 -20726.083,E2 -20726.083} C_VEL
LIN {X 0,Y 278.821,Z 531.113,A -85,B 0,C 180,E1 -20726.851,E2 -20726.851} C_VEL
LIN {X 0,Y 274.855,Z 547.274,A -85,B 0,C 180,E1 -20727.9,E2 -20727.9} C_VEL
LIN {X 0,Y 270.483,Z 561.856,A -85,B 0,C 180,E1 -20729.11,E2 -20729.11} C_VEL
LIN {X 0,Y 265.328,Z 576.232,A -85,B 0,C 180,E1 -20730.608,E2 -20730.608} C_VEL
LIN {X 0,Y 259.914,Z 589.508,A -85,B 0,C 180,E1 -20732.328,E2 -20732.328} C_VEL
LIN {X 0,Y 254.128,Z 602.012,A -85,B 0,C 180,E1 -20734.289,E2 -20734.289} C_VEL
LIN {X 0,Y 247.987,Z 614.151,A -85,B 0,C 180,E1 -20736.65,E2 -20736.65} C_VEL
LIN {X 0,Y 241.381,Z 625.901,A -85,B 0,C 180,E1 -20739.489,E2 -20739.489} C_VEL
LIN {X 0,Y 235.503,Z 635.549,A -85,B 0,C 180,E1 -20742.387,E2 -20742.387} C_VEL
LIN {X 0,Y 229.612,Z 644.803,A -85,B 0,C 180,E1 -20745.866,E2 -20745.866} C_VEL
LIN {X 0,Y 225.2,Z 651.613,A -85,B 0,C 180,E1 -20749.052,E2 -20749.052} C_VEL
LIN {X 0,Y 220.892,Z 657.941,A -85,B 0,C 180,E1 -20752.806,E2 -20752.806} C_VEL
LIN {X 0,Y 217.449,Z 662.994,A -85,B 0,C 180,E1 -20756.671,E2 -20756.671} C_VEL
LIN {X 0,Y 214.821,Z 666.899,A -85,B 0,C 180,E1 -20760.611,E2 -20760.611} C_VEL
LIN {X 0,Y 213.011,Z 669.587,A -85,B 0,C 180,E1 -20764.601,E2 -20764.601} C_VEL
LIN {X 0,Y 211.893,Z 671.27,A -85,B 0,C 180,E1 -20768.602,E2 -20768.602} C_VEL
LIN {X 0,Y 211.295,Z 671.892,A -85,B 0,C 180,E1 -20772.581,E2 -20772.581} C_VEL
LIN {X 0,Y 211.14,Z 671.526,A -85,B 0,C 180,E1 -20776.526,E2 -20776.526} C_VEL
LIN {X 0,Y 211.194,Z 670.187,A -85,B 0,C 180,E1 -20780.422,E2 -20780.422} C_VEL
LIN {X 0,Y 211.785,Z 667.6,A -85,B 0,C 180,E1 -20784.596,E2 -20784.596} C_VEL
LIN {X 0,Y 212.29,Z 664.545,A -85,B 0,C 180,E1 -20788.103,E2 -20788.103} C_VEL
LIN {X 0,Y 213.458,Z 660.143,A -85,B 0,C 180,E1 -20791.887,E2 -20791.887} C_VEL
LIN {X 0,Y 215.126,Z 654.715,A -85,B 0,C 180,E1 -20795.624,E2 -20795.624} C_VEL
LIN {X 0,Y 217.561,Z 647.987,A -85,B 0,C 180,E1 -20799.295,E2 -20799.295} C_VEL
LIN {X 0,Y 220.739,Z 639.922,A -85,B 0,C 180,E1 -20802.877,E2 -20802.877} C_VEL
LIN {X 0,Y 224.646,Z 630.328,A -85,B 0,C 180,E1 -20806.353,E2 -20806.353} C_VEL
LIN {X 0,Y 228.548,Z 620.467,A -85,B 0,C 180,E1 -20809.303,E2 -20809.303} C_VEL
LIN {X 0,Y 232.904,Z 608.858,A -85,B 0,C 180,E1 -20812.16,E2 -20812.16} C_VEL
LIN {X 0,Y 237.314,Z 596.209,A -85,B 0,C 180,E1 -20814.728,E2 -20814.728} C_VEL
LIN {X 0,Y 241.355,Z 583.691,A -85,B 0,C 180,E1 -20816.83,E2 -20816.83} C_VEL
LIN {X 0,Y 245.369,Z 570.259,A -85,B 0,C 180,E1 -20818.67,E2 -20818.67} C_VEL
LIN {X 0,Y 249.025,Z 555.775,A -85,B 0,C 180,E1 -20820.296,E2 -20820.296} C_VEL
LIN {X 0,Y 252.216,Z 541.12,A -85,B 0,C 180,E1 -20821.615,E2 -20821.615} C_VEL
LIN {X 0,Y 255.219,Z 525.071,A -85,B 0,C 180,E1 -20822.712,E2 -20822.712} C_VEL
LIN {X 0,Y 257.527,Z 508.57,A -85,B 0,C 180,E1 -20823.547,E2 -20823.547} C_VEL
LIN {X 0,Y 259.159,Z 491.025,A -85,B 0,C 180,E1 -20824.126,E2 -20824.126} C_VEL
LIN {X 0,Y 265.456,Z 385.39,A -85,B 0,C 180,E1 -20826.778,E2 -20826.778} C_VEL
LIN {X 0,Y 258.014,Z 371.261,A -85,B 0,C 180,E1 -20829.012,E2 -20829.012} C_VEL
LIN {X 0,Y 250.847,Z 358.955,A -85,B 0,C 180,E1 -20831.327,E2 -20831.327} C_VEL
LIN {X 0,Y 244.087,Z 348.423,A -85,B 0,C 180,E1 -20833.687,E2 -20833.687} C_VEL
LIN {X 0,Y 236.8,Z 337.918,A -85,B 0,C 180,E1 -20836.492,E2 -20836.492} C_VEL
LIN {X 0,Y 232.454,Z 332.29,A -85,B 0,C 180,E1 -20838.305,E2 -20838.305} C_VEL
LIN {X 0,Y 229.663,Z 328.563,A -85,B 0,C 180,E1 -20839.561,E2 -20839.561} C_VEL
LIN {X 0,Y 226.93,Z 324.875,A -85,B 0,C 180,E1 -20840.866,E2 -20840.866} C_VEL
LIN {X 0,Y 223.661,Z 321.049,A -85,B 0,C 180,E1 -20842.495,E2 -20842.495} C_VEL
LIN {X 0,Y 222.524,Z 319.212,A -85,B 0,C 180,E1 -20843.123,E2 -20843.123} C_VEL
LIN {X 0,Y 219.871,Z 316.756,A -85,B 0,C 180,E1 -20844.537,E2 -20844.537} C_VEL
LIN {X 0,Y 218.142,Z 313.818,A -85,B 0,C 180,E1 -20845.61,E2 -20845.61} C_VEL
LIN {X 0,Y 215.668,Z 312.151,A -85,B 0,C 180,E1 -20847.056,E2 -20847.056} C_VEL
LIN {X 0,Y 214.21,Z 309.962,A -85,B 0,C 180,E1 -20848.058,E2 -20848.058} C_VEL
LIN {X 0,Y 213.761,Z 308.17,A -85,B 0,C 180,E1 -20848.506,E2 -20848.506} C_VEL
LIN {X 0,Y 213.787,Z 308.157,A -85,B 0,C 180,E1 -20852.597,E2 -20852.597} C_VEL
LIN {X 0,Y 213.812,Z 308.142,A -85,B 0,C 180,E1 -20856.979,E2 -20856.979} C_VEL
LIN {X 0,Y 213.888,Z 308.13,A -85,B 0,C 180,E1 -20862.343,E2 -20862.343} C_VEL
LIN {X 0,Y 213.944,Z 308.13,A -85,B 0,C 180,E1 -20866.705,E2 -20866.705} C_VEL
LIN {X 0,Y 214.14,Z 308.119,A -85,B 0,C 180,E1 -20870.554,E2 -20870.554} C_VEL
LIN {X 0,Y 214.088,Z 308.103,A -85,B 0,C 180,E1 -20874.347,E2 -20874.347} C_VEL
LIN {X 0,Y 214.478,Z 308.059,A -85,B 0,C 180,E1 -20879.28,E2 -20879.28} C_VEL
LIN {X 0,Y 214.445,Z 308.067,A -85,B 0,C 180,E1 -20881.877,E2 -20881.877} C_VEL
LIN {X 0,Y 214.175,Z 308.08,A -85,B 0,C 180,E1 -20887.336,E2 -20887.336} C_VEL
LIN {X 0,Y 213.539,Z 308.168,A -85,B 0,C 180,E1 -20888.379,E2 -20888.379} C_VEL
LIN {X 0,Y 210.602,Z 308.558,A -85,B 0,C 180,E1 -20890.009,E2 -20890.009} C_VEL
LIN {X 0,Y 207.59,Z 308.935,A -85,B 0,C 180,E1 -20891.684,E2 -20891.684} C_VEL
LIN {X 0,Y 206.892,Z 309.019,A -85,B 0,C 180,E1 -20892.78,E2 -20892.78} C_VEL
LIN {X 0,Y 206.915,Z 309.183,A -85,B 0,C 180,E1 -20893.628,E2 -20893.628} C_VEL
LIN {X 0,Y 207.568,Z 311.327,A -85,B 0,C 180,E1 -20894.334,E2 -20894.334} C_VEL
LIN {X 0,Y 209.524,Z 313.722,A -85,B 0,C 180,E1 -20895.939,E2 -20895.939} C_VEL
LIN {X 0,Y 211.765,Z 315.07,A -85,B 0,C 180,E1 -20897.501,E2 -20897.501} C_VEL
LIN {X 0,Y 213.236,Z 317.96,A -85,B 0,C 180,E1 -20898.619,E2 -20898.619} C_VEL
LIN {X 0,Y 215.637,Z 320.156,A -85,B 0,C 180,E1 -20900.135,E2 -20900.135} C_VEL
LIN {X 0,Y 216.43,Z 320.902,A -85,B 0,C 180,E1 -20900.616,E2 -20900.616} C_VEL
LIN {X 0,Y 218.671,Z 324.22,A -85,B 0,C 180,E1 -20902,E2 -20902} C_VEL
LIN {X 0,Y 220.744,Z 326.259,A -85,B 0,C 180,E1 -20903.135,E2 -20903.135} C_VEL
LIN {X 0,Y 223.433,Z 329.853,A -85,B 0,C 180,E1 -20904.58,E2 -20904.58} C_VEL
LIN {X 0,Y 224.93,Z 331.73,A -85,B 0,C 180,E1 -20905.336,E2 -20905.336} C_VEL
LIN {X 0,Y 228.751,Z 336.764,A -85,B 0,C 180,E1 -20907.168,E2 -20907.168} C_VEL
LIN {X 0,Y 234.978,Z 345.289,A -85,B 0,C 180,E1 -20909.89,E2 -20909.89} C_VEL
LIN {X 0,Y 241.24,Z 354.536,A -85,B 0,C 180,E1 -20912.364,E2 -20912.364} C_VEL
LIN {X 0,Y 247.428,Z 366.045,A -85,B 0,C 180,E1 -20914.678,E2 -20914.678} C_VEL
LIN {X 0,Y 253.229,Z 377.761,A -85,B 0,C 180,E1 -20916.703,E2 -20916.703} C_VEL
LIN {X 0,Y 259.502,Z 392.041,A -85,B 0,C 180,E1 -20918.776,E2 -20918.776} C_VEL
LIN {X 0,Y 260.185,Z 393.726,A -85,B 0,C 180,E1 -20918.996,E2 -20918.996} C_VEL
LIN {X 0,Y 252.981,Z 508.6,A -85,B 0,C 180,E1 -20921.93,E2 -20921.93} C_VEL
LIN {X 0,Y 251.023,Z 525.431,A -85,B 0,C 180,E1 -20922.594,E2 -20922.594} C_VEL
LIN {X 0,Y 248.249,Z 541.758,A -85,B 0,C 180,E1 -20923.494,E2 -20923.494} C_VEL
LIN {X 0,Y 245.041,Z 557.056,A -85,B 0,C 180,E1 -20924.631,E2 -20924.631} C_VEL
LIN {X 0,Y 241.533,Z 571.319,A -85,B 0,C 180,E1 -20925.997,E2 -20925.997} C_VEL
LIN {X 0,Y 237.717,Z 584.261,A -85,B 0,C 180,E1 -20927.509,E2 -20927.509} C_VEL
LIN {X 0,Y 233.555,Z 597.473,A -85,B 0,C 180,E1 -20929.404,E2 -20929.404} C_VEL
LIN {X 0,Y 229.071,Z 610.058,A -85,B 0,C 180,E1 -20931.591,E2 -20931.591} C_VEL
LIN {X 0,Y 224.674,Z 621.771,A -85,B 0,C 180,E1 -20934.08,E2 -20934.08} C_VEL
LIN {X 0,Y 220.053,Z 633.544,A -85,B 0,C 180,E1 -20937.116,E2 -20937.116} C_VEL
LIN {X 0,Y 215.985,Z 643.574,A -85,B 0,C 180,E1 -20940.25,E2 -20940.25} C_VEL
LIN {X 0,Y 212.497,Z 652.455,A -85,B 0,C 180,E1 -20943.657,E2 -20943.657} C_VEL
LIN {X 0,Y 209.492,Z 660.306,A -85,B 0,C 180,E1 -20947.307,E2 -20947.307} C_VEL
LIN {X 0,Y 207.172,Z 667.155,A -85,B 0,C 180,E1 -20951.2,E2 -20951.2} C_VEL
LIN {X 0,Y 205.631,Z 672.659,A -85,B 0,C 180,E1 -20955.148,E2 -20955.148} C_VEL
LIN {X 0,Y 204.831,Z 676.057,A -85,B 0,C 180,E1 -20958.12,E2 -20958.12} C_VEL
LIN {X 0,Y 204.407,Z 679.554,A -85,B 0,C 180,E1 -20962.095,E2 -20962.095} C_VEL
LIN {X 0,Y 204.361,Z 682.065,A -85,B 0,C 180,E1 -20966.056,E2 -20966.056} C_VEL
LIN {X 0,Y 204.478,Z 683.461,A -85,B 0,C 180,E1 -20970,E2 -20970} C_VEL
LIN {X 0,Y 204.317,Z 683.946,A -85,B 0,C 180,E1 -20974.045,E2 -20974.045} C_VEL
LIN {X 0,Y 204.371,Z 683.379,A -85,B 0,C 180,E1 -20977.907,E2 -20977.907} C_VEL
LIN {X 0,Y 204.9,Z 681.947,A -85,B 0,C 180,E1 -20981.876,E2 -20981.876} C_VEL
LIN {X 0,Y 206.166,Z 679.483,A -85,B 0,C 180,E1 -20985.826,E2 -20985.826} C_VEL
LIN {X 0,Y 208.167,Z 676.115,A -85,B 0,C 180,E1 -20989.732,E2 -20989.732} C_VEL
LIN {X 0,Y 211.864,Z 670.386,A -85,B 0,C 180,E1 -20994.498,E2 -20994.498} C_VEL
LIN {X 0,Y 216.255,Z 663.698,A -85,B 0,C 180,E1 -20998.664,E2 -20998.664} C_VEL
LIN {X 0,Y 221.771,Z 655.525,A -85,B 0,C 180,E1 -21002.598,E2 -21002.598} C_VEL
LIN {X 0,Y 227.544,Z 646.762,A -85,B 0,C 180,E1 -21005.933,E2 -21005.933} C_VEL
LIN {X 0,Y 233.028,Z 637.906,A -85,B 0,C 180,E1 -21008.687,E2 -21008.687} C_VEL
LIN {X 0,Y 239.233,Z 627.266,A -85,B 0,C 180,E1 -21011.376,E2 -21011.376} C_VEL
LIN {X 0,Y 246.06,Z 614.983,A -85,B 0,C 180,E1 -21013.839,E2 -21013.839} C_VEL
LIN {X 0,Y 252.329,Z 602.231,A -85,B 0,C 180,E1 -21015.943,E2 -21015.943} C_VEL
LIN {X 0,Y 258.653,Z 588.116,A -85,B 0,C 180,E1 -21017.768,E2 -21017.768} C_VEL
LIN {X 0,Y 264.261,Z 573.476,A -85,B 0,C 180,E1 -21019.285,E2 -21019.285} C_VEL
LIN {X 0,Y 268.855,Z 559.418,A -85,B 0,C 180,E1 -21020.457,E2 -21020.457} C_VEL
LIN {X 0,Y 273.059,Z 544.424,A -85,B 0,C 180,E1 -21021.425,E2 -21021.425} C_VEL
LIN {X 0,Y 276.77,Z 527.563,A -85,B 0,C 180,E1 -21022.242,E2 -21022.242} C_VEL
LIN {X 0,Y 279.391,Z 510.793,A -85,B 0,C 180,E1 -21022.808,E2 -21022.808} C_VEL
LIN {X 0,Y 281.828,Z 482.346,A -85,B 0,C 180,E1 -21023.503,E2 -21023.503} C_VEL
LIN {X 0,Y 287.288,Z 411.312,A -85,B 0,C 180,E1 -21025.138,E2 -21025.138} C_VEL
LIN {X 0,Y 282.969,Z 402.115,A -85,B 0,C 180,E1 -21027.208,E2 -21027.208} C_VEL
LIN {X 0,Y 277.428,Z 391.265,A -85,B 0,C 180,E1 -21030.176,E2 -21030.176} C_VEL
LIN {X 0,Y 274.383,Z 385.962,A -85,B 0,C 180,E1 -21031.976,E2 -21031.976} C_VEL
LIN {X 0,Y 270.565,Z 379.333,A -85,B 0,C 180,E1 -21034.517,E2 -21034.517} C_VEL
LIN {X 0,Y 268.811,Z 376.747,A -85,B 0,C 180,E1 -21035.797,E2 -21035.797} C_VEL
LIN {X 0,Y 266.172,Z 372.9,A -85,B 0,C 180,E1 -21037.936,E2 -21037.936} C_VEL
LIN {X 0,Y 263.58,Z 369.23,A -85,B 0,C 180,E1 -21040.403,E2 -21040.403} C_VEL
LIN {X 0,Y 260.343,Z 364.766,A -85,B 0,C 180,E1 -21044.456,E2 -21044.456} C_VEL
LIN {X 0,Y 259.836,Z 363.687,A -85,B 0,C 180,E1 -21045.345,E2 -21045.345} C_VEL
LIN {X 0,Y 257.374,Z 361.038,A -85,B 0,C 180,E1 -21052.154,E2 -21052.154} C_VEL
LIN {X 0,Y 257.291,Z 360.899,A -85,B 0,C 180,E1 -21054.243,E2 -21054.243} C_VEL
LIN {X 0,Y 258.204,Z 362.069,A -85,B 0,C 180,E1 -21058.771,E2 -21058.771} C_VEL
LIN {X 0,Y 260.228,Z 364.028,A -85,B 0,C 180,E1 -21062.71,E2 -21062.71} C_VEL
LIN {X 0,Y 262.53,Z 367.767,A -85,B 0,C 180,E1 -21065.895,E2 -21065.895} C_VEL
LIN {X 0,Y 263.62,Z 369.072,A -85,B 0,C 180,E1 -21067.059,E2 -21067.059} C_VEL
LIN {X 0,Y 266.23,Z 372.838,A -85,B 0,C 180,E1 -21069.545,E2 -21069.545} C_VEL
LIN {X 0,Y 270.357,Z 378.874,A -85,B 0,C 180,E1 -21072.77,E2 -21072.77} C_VEL
LIN {X 0,Y 273.082,Z 382.967,A -85,B 0,C 180,E1 -21074.593,E2 -21074.593} C_VEL
LIN {X 0,Y 277.769,Z 390.15,A -85,B 0,C 180,E1 -21077.355,E2 -21077.355} C_VEL
LIN {X 0,Y 283.498,Z 399.661,A -85,B 0,C 180,E1 -21080.309,E2 -21080.309} C_VEL
LIN {X 0,Y 287.531,Z 406.865,A -85,B 0,C 180,E1 -21082.169,E2 -21082.169} C_VEL
LIN {X 0,Y 280.197,Z 500.224,A -85,B 0,C 180,E1 -21084.347,E2 -21084.347} C_VEL
LIN {X 0,Y 277.642,Z 517.18,A -85,B 0,C 180,E1 -21084.916,E2 -21084.916} C_VEL
LIN {X 0,Y 274.689,Z 532.118,A -85,B 0,C 180,E1 -21085.679,E2 -21085.679} C_VEL
LIN {X 0,Y 270.531,Z 548.356,A -85,B 0,C 180,E1 -21086.745,E2 -21086.745} C_VEL
LIN {X 0,Y 266.309,Z 561.896,A -85,B 0,C 180,E1 -21087.861,E2 -21087.861} C_VEL
LIN {X 0,Y 260.754,Z 576.965,A -85,B 0,C 180,E1 -21089.435,E2 -21089.435} C_VEL
LIN {X 0,Y 254.865,Z 590.831,A -85,B 0,C 180,E1 -21091.258,E2 -21091.258} C_VEL
LIN {X 0,Y 248.897,Z 603.143,A -85,B 0,C 180,E1 -21093.226,E2 -21093.226} C_VEL
LIN {X 0,Y 243.396,Z 613.614,A -85,B 0,C 180,E1 -21095.276,E2 -21095.276} C_VEL
LIN {X 0,Y 237.56,Z 623.753,A -85,B 0,C 180,E1 -21097.685,E2 -21097.685} C_VEL
LIN {X 0,Y 231.325,Z 633.77,A -85,B 0,C 180,E1 -21100.576,E2 -21100.576} C_VEL
LIN {X 0,Y 225.891,Z 642.002,A -85,B 0,C 180,E1 -21103.515,E2 -21103.515} C_VEL
LIN {X 0,Y 220.991,Z 649.137,A -85,B 0,C 180,E1 -21106.664,E2 -21106.664} C_VEL
LIN {X 0,Y 215.962,Z 656.271,A -85,B 0,C 180,E1 -21110.611,E2 -21110.611} C_VEL
LIN {X 0,Y 211.986,Z 661.747,A -85,B 0,C 180,E1 -21114.536,E2 -21114.536} C_VEL
LIN {X 0,Y 209.618,Z 665.041,A -85,B 0,C 180,E1 -21117.558,E2 -21117.558} C_VEL
LIN {X 0,Y 206.997,Z 668.62,A -85,B 0,C 180,E1 -21121.979,E2 -21121.979} C_VEL
LIN {X 0,Y 205.492,Z 670.648,A -85,B 0,C 180,E1 -21125.769,E2 -21125.769} C_VEL
LIN {X 0,Y 204.518,Z 671.879,A -85,B 0,C 180,E1 -21129.901,E2 -21129.901} C_VEL
LIN {X 0,Y 204.125,Z 672.003,A -85,B 0,C 180,E1 -21134.592,E2 -21134.592} C_VEL
LIN {X 0,Y 204.02,Z 671.302,A -85,B 0,C 180,E1 -21138.072,E2 -21138.072} C_VEL
LIN {X 0,Y 204.25,Z 669.497,A -85,B 0,C 180,E1 -21142.089,E2 -21142.089} C_VEL
LIN {X 0,Y 204.879,Z 666.786,A -85,B 0,C 180,E1 -21146.066,E2 -21146.066} C_VEL
LIN {X 0,Y 206.038,Z 661.91,A -85,B 0,C 180,E1 -21150.977,E2 -21150.977} C_VEL
LIN {X 0,Y 208.072,Z 655.348,A -85,B 0,C 180,E1 -21155.816,E2 -21155.816} C_VEL
LIN {X 0,Y 210.588,Z 648.701,A -85,B 0,C 180,E1 -21159.605,E2 -21159.605} C_VEL
LIN {X 0,Y 213.844,Z 640.753,A -85,B 0,C 180,E1 -21163.3,E2 -21163.3} C_VEL
LIN {X 0,Y 217.9,Z 631.283,A -85,B 0,C 180,E1 -21166.875,E2 -21166.875} C_VEL
LIN {X 0,Y 221.904,Z 621.491,A -85,B 0,C 180,E1 -21169.905,E2 -21169.905} C_VEL
LIN {X 0,Y 226.419,Z 610.035,A -85,B 0,C 180,E1 -21172.83,E2 -21172.83} C_VEL
LIN {X 0,Y 230.941,Z 597.584,A -85,B 0,C 180,E1 -21175.458,E2 -21175.458} C_VEL
LIN {X 0,Y 235.516,Z 584.03,A -85,B 0,C 180,E1 -21177.792,E2 -21177.792} C_VEL
LIN {X 0,Y 239.662,Z 570.612,A -85,B 0,C 180,E1 -21179.66,E2 -21179.66} C_VEL
LIN {X 0,Y 243.442,Z 556.163,A -85,B 0,C 180,E1 -21181.308,E2 -21181.308} C_VEL
LIN {X 0,Y 246.736,Z 541.559,A -85,B 0,C 180,E1 -21182.643,E2 -21182.643} C_VEL
LIN {X 0,Y 249.83,Z 525.592,A -85,B 0,C 180,E1 -21183.751,E2 -21183.751} C_VEL
LIN {X 0,Y 252.198,Z 509.174,A -85,B 0,C 180,E1 -21184.596,E2 -21184.596} C_VEL
LIN {X 0,Y 253.894,Z 491.845,A -85,B 0,C 180,E1 -21185.177,E2 -21185.177} C_VEL
LIN {X 0,Y 260.338,Z 388.224,A -85,B 0,C 180,E1 -21187.797,E2 -21187.797} C_VEL
LIN {X 0,Y 253.516,Z 375.107,A -85,B 0,C 180,E1 -21189.952,E2 -21189.952} C_VEL
LIN {X 0,Y 246.647,Z 363.154,A -85,B 0,C 180,E1 -21192.278,E2 -21192.278} C_VEL
LIN {X 0,Y 239.245,Z 351.525,A -85,B 0,C 180,E1 -21195.014,E2 -21195.014} C_VEL
LIN {X 0,Y 232.78,Z 342.395,A -85,B 0,C 180,E1 -21197.641,E2 -21197.641} C_VEL
LIN {X 0,Y 229.585,Z 338.075,A -85,B 0,C 180,E1 -21199.05,E2 -21199.05} C_VEL
LIN {X 0,Y 226.947,Z 334.511,A -85,B 0,C 180,E1 -21200.286,E2 -21200.286} C_VEL
LIN {X 0,Y 223.614,Z 330.119,A -85,B 0,C 180,E1 -21201.943,E2 -21201.943} C_VEL
LIN {X 0,Y 220.794,Z 326.426,A -85,B 0,C 180,E1 -21203.446,E2 -21203.446} C_VEL
LIN {X 0,Y 219.91,Z 325.337,A -85,B 0,C 180,E1 -21203.934,E2 -21203.934} C_VEL
LIN {X 0,Y 217.188,Z 322.33,A -85,B 0,C 180,E1 -21205.491,E2 -21205.491} C_VEL
LIN {X 0,Y 216.115,Z 320.413,A -85,B 0,C 180,E1 -21206.192,E2 -21206.192} C_VEL
LIN {X 0,Y 213.672,Z 318.538,A -85,B 0,C 180,E1 -21207.69,E2 -21207.69} C_VEL
LIN {X 0,Y 211.874,Z 315.692,A -85,B 0,C 180,E1 -21208.994,E2 -21208.994} C_VEL
LIN {X 0,Y 211.461,Z 314.876,A -85,B 0,C 180,E1 -21209.32,E2 -21209.32} C_VEL
LIN {X 0,Y 208.733,Z 313.196,A -85,B 0,C 180,E1 -21211.271,E2 -21211.271} C_VEL
LIN {X 0,Y 207.239,Z 310.906,A -85,B 0,C 180,E1 -21212.569,E2 -21212.569} C_VEL
LIN {X 0,Y 206.739,Z 309.045,A -85,B 0,C 180,E1 -21213.227,E2 -21213.227} C_VEL
LIN {X 0,Y 206.735,Z 309.033,A -85,B 0,C 180,E1 -21218.04,E2 -21218.04} C_VEL
LIN {X 0,Y 206.827,Z 309.008,A -85,B 0,C 180,E1 -21222.191,E2 -21222.191} C_VEL
LIN {X 0,Y 206.884,Z 309.015,A -85,B 0,C 180,E1 -21226.242,E2 -21226.242} C_VEL
LIN {X 0,Y 207.1,Z 308.99,A -85,B 0,C 180,E1 -21230.23,E2 -21230.23} C_VEL
LIN {X 0,Y 207.051,Z 308.979,A -85,B 0,C 180,E1 -21234.154,E2 -21234.154} C_VEL
LIN {X 0,Y 207.376,Z 308.96,A -85,B 0,C 180,E1 -21238.057,E2 -21238.057} C_VEL
LIN {X 0,Y 207.511,Z 308.922,A -85,B 0,C 180,E1 -21239.999,E2 -21239.999} C_VEL
LIN {X 0,Y 207.382,Z 308.947,A -85,B 0,C 180,E1 -21241.941,E2 -21241.941} C_VEL
LIN {X 0,Y 207.139,Z 308.957,A -85,B 0,C 180,E1 -21247.799,E2 -21247.799} C_VEL
LIN {X 0,Y 206.921,Z 309.017,A -85,B 0,C 180,E1 -21251.757,E2 -21251.757} C_VEL
LIN {X 0,Y 206.892,Z 309.019,A -85,B 0,C 180,E1 -21252.78,E2 -21252.78} C_VEL
LIN {X 0,Y 207.117,Z 309.773,A -85,B 0,C 180,E1 -21253.628,E2 -21253.628} C_VEL
LIN {X 0,Y 207.824,Z 312.454,A -85,B 0,C 180,E1 -21254.632,E2 -21254.632} C_VEL
LIN {X 0,Y 209.715,Z 321.378,A -85,B 0,C 180,E1 -21256.742,E2 -21256.742} C_VEL
LIN {X 0,Y 210.233,Z 322.642,A -85,B 0,C 180,E1 -21257.184,E2 -21257.184} C_VEL
LIN {X 0,Y 212.44,Z 325.666,A -85,B 0,C 180,E1 -21258.769,E2 -21258.769} C_VEL
LIN {X 0,Y 214.371,Z 327.44,A -85,B 0,C 180,E1 -21259.993,E2 -21259.993} C_VEL
LIN {X 0,Y 216.868,Z 330.912,A -85,B 0,C 180,E1 -21261.568,E2 -21261.568} C_VEL
LIN {X 0,Y 218.684,Z 332.908,A -85,B 0,C 180,E1 -21262.605,E2 -21262.605} C_VEL
LIN {X 0,Y 221.619,Z 336.622,A -85,B 0,C 180,E1 -21264.21,E2 -21264.21} C_VEL
LIN {X 0,Y 226.099,Z 342.79,A -85,B 0,C 180,E1 -21266.477,E2 -21266.477} C_VEL
LIN {X 0,Y 229.875,Z 348.05,A -85,B 0,C 180,E1 -21268.224,E2 -21268.224} C_VEL
LIN {X 0,Y 236.264,Z 357.285,A -85,B 0,C 180,E1 -21270.933,E2 -21270.933} C_VEL
LIN {X 0,Y 241.021,Z 365.728,A -85,B 0,C 180,E1 -21272.831,E2 -21272.831} C_VEL
LIN {X 0,Y 248.027,Z 379.845,A -85,B 0,C 180,E1 -21275.449,E2 -21275.449} C_VEL
LIN {X 0,Y 254.036,Z 393.477,A -85,B 0,C 180,E1 -21277.552,E2 -21277.552} C_VEL
LIN {X 0,Y 255.073,Z 395.966,A -85,B 0,C 180,E1 -21277.903,E2 -21277.903} C_VEL
LIN {X 0,Y 247.769,Z 509.254,A -85,B 0,C 180,E1 -21280.837,E2 -21280.837} C_VEL
LIN {X 0,Y 245.648,Z 526.439,A -85,B 0,C 180,E1 -21281.536,E2 -21281.536} C_VEL
LIN {X 0,Y 242.82,Z 542.297,A -85,B 0,C 180,E1 -21282.434,E2 -21282.434} C_VEL
LIN {X 0,Y 239.519,Z 557.419,A -85,B 0,C 180,E1 -21283.582,E2 -21283.582} C_VEL
LIN {X 0,Y 235.395,Z 573.274,A -85,B 0,C 180,E1 -21285.142,E2 -21285.142} C_VEL
LIN {X 0,Y 230.75,Z 588.314,A -85,B 0,C 180,E1 -21287.003,E2 -21287.003} C_VEL
LIN {X 0,Y 225.961,Z 602.398,A -85,B 0,C 180,E1 -21289.22,E2 -21289.22} C_VEL
LIN {X 0,Y 221.139,Z 615.235,A -85,B 0,C 180,E1 -21291.704,E2 -21291.704} C_VEL
LIN {X 0,Y 215.994,Z 627.94,A -85,B 0,C 180,E1 -21294.722,E2 -21294.722} C_VEL
LIN {X 0,Y 211.489,Z 638.737,A -85,B 0,C 180,E1 -21297.88,E2 -21297.88} C_VEL
LIN {X 0,Y 207.592,Z 647.963,A -85,B 0,C 180,E1 -21301.156,E2 -21301.156} C_VEL
LIN {X 0,Y 204.008,Z 656.835,A -85,B 0,C 180,E1 -21305.039,E2 -21305.039} C_VEL
LIN {X 0,Y 201.469,Z 663.391,A -85,B 0,C 180,E1 -21308.514,E2 -21308.514} C_VEL
LIN {X 0,Y 199.358,Z 669.816,A -85,B 0,C 180,E1 -21312.714,E2 -21312.714} C_VEL
LIN {X 0,Y 198.083,Z 674.574,A -85,B 0,C 180,E1 -21316.667,E2 -21316.667} C_VEL
LIN {X 0,Y 197.491,Z 677.566,A -85,B 0,C 180,E1 -21319.751,E2 -21319.751} C_VEL
LIN {X 0,Y 197.278,Z 680.629,A -85,B 0,C 180,E1 -21323.865,E2 -21323.865} C_VEL
LIN {X 0,Y 197.272,Z 682.599,A -85,B 0,C 180,E1 -21327.959,E2 -21327.959} C_VEL
LIN {X 0,Y 197.396,Z 683.212,A -85,B 0,C 180,E1 -21330,E2 -21330} C_VEL
LIN {X 0,Y 197.241,Z 683.727,A -85,B 0,C 180,E1 -21334.087,E2 -21334.087} C_VEL
LIN {X 0,Y 197.296,Z 683.212,A -85,B 0,C 180,E1 -21338.192,E2 -21338.192} C_VEL
LIN {X 0,Y 197.885,Z 681.808,A -85,B 0,C 180,E1 -21342.304,E2 -21342.304} C_VEL
LIN {X 0,Y 199.257,Z 679.403,A -85,B 0,C 180,E1 -21346.39,E2 -21346.39} C_VEL
LIN {X 0,Y 201.406,Z 676.065,A -85,B 0,C 180,E1 -21350.423,E2 -21350.423} C_VEL
LIN {X 0,Y 204.43,Z 671.646,A -85,B 0,C 180,E1 -21354.365,E2 -21354.365} C_VEL
LIN {X 0,Y 208.283,Z 666.211,A -85,B 0,C 180,E1 -21358.19,E2 -21358.19} C_VEL
LIN {X 0,Y 214.406,Z 657.686,A -85,B 0,C 180,E1 -21362.742,E2 -21362.742} C_VEL
LIN {X 0,Y 220.201,Z 649.311,A -85,B 0,C 180,E1 -21366.189,E2 -21366.189} C_VEL
LIN {X 0,Y 226.705,Z 639.406,A -85,B 0,C 180,E1 -21369.458,E2 -21369.458} C_VEL
LIN {X 0,Y 233.957,Z 627.655,A -85,B 0,C 180,E1 -21372.524,E2 -21372.524} C_VEL
LIN {X 0,Y 240.999,Z 615.49,A -85,B 0,C 180,E1 -21375.006,E2 -21375.006} C_VEL
LIN {X 0,Y 247.394,Z 603.049,A -85,B 0,C 180,E1 -21377.09,E2 -21377.09} C_VEL
LIN {X 0,Y 253.968,Z 588.867,A -85,B 0,C 180,E1 -21378.946,E2 -21378.946} C_VEL
LIN {X 0,Y 259.733,Z 574.452,A -85,B 0,C 180,E1 -21380.459,E2 -21380.459} C_VEL
LIN {X 0,Y 264.449,Z 560.703,A -85,B 0,C 180,E1 -21381.628,E2 -21381.628} C_VEL
LIN {X 0,Y 269.064,Z 544.887,A -85,B 0,C 180,E1 -21382.659,E2 -21382.659} C_VEL
LIN {X 0,Y 272.96,Z 527.685,A -85,B 0,C 180,E1 -21383.491,E2 -21383.491} C_VEL
LIN {X 0,Y 275.673,Z 510.933,A -85,B 0,C 180,E1 -21384.051,E2 -21384.051} C_VEL
LIN {X 0,Y 277.961,Z 485.527,A -85,B 0,C 180,E1 -21384.678,E2 -21384.678} C_VEL
LIN {X 0,Y 283.585,Z 414.623,A -85,B 0,C 180,E1 -21386.305,E2 -21386.305} C_VEL
LIN {X 0,Y 278.861,Z 404.528,A -85,B 0,C 180,E1 -21388.746,E2 -21388.746} C_VEL
LIN {X 0,Y 274.081,Z 395.15,A -85,B 0,C 180,E1 -21391.511,E2 -21391.511} C_VEL
LIN {X 0,Y 269.927,Z 387.748,A -85,B 0,C 180,E1 -21394.239,E2 -21394.239} C_VEL
LIN {X 0,Y 267.482,Z 383.632,A -85,B 0,C 180,E1 -21396.071,E2 -21396.071} C_VEL
LIN {X 0,Y 264.806,Z 379.668,A -85,B 0,C 180,E1 -21398.304,E2 -21398.304} C_VEL
LIN {X 0,Y 262.153,Z 375.724,A -85,B 0,C 180,E1 -21400.945,E2 -21400.945} C_VEL
LIN {X 0,Y 259.389,Z 371.975,A -85,B 0,C 180,E1 -21404.515,E2 -21404.515} C_VEL
LIN {X 0,Y 258.804,Z 370.675,A -85,B 0,C 180,E1 -21405.57,E2 -21405.57} C_VEL
LIN {X 0,Y 256.427,Z 367.941,A -85,B 0,C 180,E1 -21413.042,E2 -21413.042} C_VEL
LIN {X 0,Y 256.962,Z 368.673,A -85,B 0,C 180,E1 -21417.65,E2 -21417.65} C_VEL
LIN {X 0,Y 259.134,Z 370.936,A -85,B 0,C 180,E1 -21422.403,E2 -21422.403} C_VEL
LIN {X 0,Y 261.493,Z 374.797,A -85,B 0,C 180,E1 -21425.753,E2 -21425.753} C_VEL
LIN {X 0,Y 262.377,Z 375.937,A -85,B 0,C 180,E1 -21426.731,E2 -21426.731} C_VEL
LIN {X 0,Y 265.535,Z 380.636,A -85,B 0,C 180,E1 -21429.775,E2 -21429.775} C_VEL
LIN {X 0,Y 268.714,Z 385.449,A -85,B 0,C 180,E1 -21432.301,E2 -21432.301} C_VEL
LIN {X 0,Y 271.601,Z 389.912,A -85,B 0,C 180,E1 -21434.297,E2 -21434.297} C_VEL
LIN {X 0,Y 276.036,Z 396.952,A -85,B 0,C 180,E1 -21436.985,E2 -21436.985} C_VEL
LIN {X 0,Y 281.282,Z 405.939,A -85,B 0,C 180,E1 -21439.779,E2 -21439.779} C_VEL
LIN {X 0,Y 283.817,Z 410.577,A -85,B 0,C 180,E1 -21441.013,E2 -21441.013} C_VEL
LIN {X 0,Y 276.576,Z 499.926,A -85,B 0,C 180,E1 -21443.089,E2 -21443.089} C_VEL
LIN {X 0,Y 274.006,Z 516.652,A -85,B 0,C 180,E1 -21443.63,E2 -21443.63} C_VEL
LIN {X 0,Y 270.708,Z 532.966,A -85,B 0,C 180,E1 -21444.456,E2 -21444.456} C_VEL
LIN {X 0,Y 266.498,Z 548.847,A -85,B 0,C 180,E1 -21445.501,E2 -21445.501} C_VEL
LIN {X 0,Y 261.678,Z 563.697,A -85,B 0,C 180,E1 -21446.746,E2 -21446.746} C_VEL
LIN {X 0,Y 256.487,Z 577.248,A -85,B 0,C 180,E1 -21448.17,E2 -21448.17} C_VEL
LIN {X 0,Y 251.033,Z 589.706,A -85,B 0,C 180,E1 -21449.786,E2 -21449.786} C_VEL
LIN {X 0,Y 244.863,Z 602.242,A -85,B 0,C 180,E1 -21451.756,E2 -21451.756} C_VEL
LIN {X 0,Y 237.987,Z 614.821,A -85,B 0,C 180,E1 -21454.221,E2 -21454.221} C_VEL
LIN {X 0,Y 231.077,Z 626.207,A -85,B 0,C 180,E1 -21457.025,E2 -21457.025} C_VEL
